(* IEC 61131-3 sources: std_i2980_v2.06_cp053/Source/IMM/ieccontrol/GlobalBaseArchives (part 4) *)

(* ---- FBGetRequiredPumps.pu ---- *)
(*
@h    ! WARNING !
@h    The Kemro K2 system (including software) only meets category B according to EN 954-1,
@h    thus it is not intended for usage in safety-relevant control applications in the field
@h    of personal safety (e.g. emergency stop).
@h    To implement potentially necessary safety-relevant control tasks, always use additional
@h    external safety devices that are intended for the particular purpose, and meet the necessary
@h    functional safety.
@h    For further information see EN 954-1 (EN ISO 13849-1) and/or the K2-x00 user manual, chapter
@h    "CE conformity, directives and standards".

get reference to the systemvariable with information about reuqired pumps for a defined movement
If the movement is not found, the reference pPumps is EMPTY.
*)

IMPORT_OVER_LISTFILE
 tsDeviceId
, tMoveIdent
, tsRequiredPumps
, tDeviceMovementList

END_IMPORT

FUNCTION_BLOCK FBGetRequiredPumps #DUMMY_EDIT_BLOCK

VAR_INPUT
 DeviceId : tsDeviceId;
 MoveDir : tMoveIdent;
 MoveId : tMoveIdent;
END_VAR

VAR_OUTPUT
 pPumps : REFTO tsRequiredPumps;
END_VAR

SYSTEM_VAR
 sv_DeviceMovements : tDeviceMovementList;
END_VAR

VAR_TEMP
 i : DINT;
 k : DINT;
END_VAR
#BEGIN_EDIT_BLOCK
(**************************************** WARNING ********************************************
 *** The KEBA Kemro K2 System including software is not intended for safety control tasks! ***
 ***                       For further information see Comment tab!                        ***
 *********************************************************************************************)

pPumps := EMPTY;

FOR i := 1 TO cMaxMoveDevicesRegistered DO
   IF (sv_DeviceMovements[i].DeviceId = DeviceId) THEN
      FOR k := 1 TO sv_DeviceMovements[i].iNumberOfMovements DO
         IF (sv_DeviceMovements[i].Movements[k]^.MoveDir = MoveDir) AND (sv_DeviceMovements[i].Movements[k]^.MoveId = MoveId) THEN
            pPumps := sv_DeviceMovements[i].Movements[k]^.AnaOutData.pRequiredPumps;
            EXIT;
         END_IF;
      END_FOR;
      EXIT;
   END_IF;
END_FOR;

;#END_EDIT_BLOCK END_FUNCTION_BLOCK

#END_OF_IEC_PART

@Puma @IecEditor 6 144 @Pou 25
@@@BEG_Comment@@@
@h    ! WARNING !
@h    The Kemro K2 system (including software) only meets category B according to EN 954-1,
@h    thus it is not intended for usage in safety-relevant control applications in the field
@h    of personal safety (e.g. emergency stop).
@h    To implement potentially necessary safety-relevant control tasks, always use additional
@h    external safety devices that are intended for the particular purpose, and meet the necessary
@h    functional safety.
@h    For further information see EN 954-1 (EN ISO 13849-1) and/or the K2-x00 user manual, chapter
@h    "CE conformity, directives and standards".

get reference to the systemvariable with information about reuqired pumps for a defined movement
If the movement is not found, the reference pPumps is EMPTY.
@@@END_Comment@@@

@BEG_Contents

@BEG_Func
@RT(17)FuncTreeContainer
0
@END_Func

@BEG_Const
@RT(18)ConstTreeContainer
0
@END_Const

@BEG_Export

@BEG_Kind
@FUNCTION_BLOCK @RT(18)FBGetRequiredPumps @STRUCTURED_TEXT
@RT(0) @RT(0) @RT(0)
@END_Kind

@BEG_Dcl
@RT(16)DclTreeContainer
7
@Var @RT(8)DeviceId @RT(0) @T @T @DERIVED 0 @T @T @DT @RT(10)tsDeviceId @RT(0) @T @T @UNKNOWN 0 @F
@F @F
@T
@BEG_Attrib
3 @RT(0) @RT(0) @RT(0)
@END_Attrib
1 1 @F @F @F @F

@Var @RT(7)MoveDir @RT(0) @T @T @DERIVED 0 @T @T @DT @RT(10)tMoveIdent @RT(0) @T @T @UNKNOWN 0 @F
@F @F
@T
@BEG_Attrib
3 @RT(0) @RT(0) @RT(0)
@END_Attrib
1 1 @F @F @F @F

@Var @RT(6)MoveId @RT(0) @T @T @DERIVED 0 @T @T @DT @RT(10)tMoveIdent @RT(0) @T @T @UNKNOWN 0 @F
@F @F
@T
@BEG_Attrib
3 @RT(0) @RT(0) @RT(0)
@END_Attrib
1 1 @F @F @F @F

@Var @RT(6)pPumps @RT(0) @T @T @REFTO 0 @F @DERIVED 0 @T @T @DT @RT(15)tsRequiredPumps @RT(0) @T @T @UNKNOWN 0 @F
@F @F
@T
@BEG_Attrib
3 @RT(0) @RT(0) @RT(0)
@END_Attrib
1 3 @F @F @F @F

@Var @RT(18)sv_DeviceMovements @RT(0) @T @T @DERIVED 0 @T @T @DT @RT(19)tDeviceMovementList @RT(0) @T @T @UNKNOWN 0 @F
@F @F
@T
@BEG_Attrib
3 @RT(0) @RT(0) @RT(0)
@END_Attrib
1 8 @F @F @F @F

@Var @RT(1)i @RT(0) @T @F @DT @RT(4)DINT @RT(0) @T @T @BASIC 0 @F
@F @F
@T
@BEG_Attrib
3 @RT(0) @RT(0) @RT(0)
@END_Attrib
1 4 @F @F @F @F

@Var @RT(1)k @RT(0) @T @F @DT @RT(4)DINT @RT(0) @T @T @BASIC 0 @F
@F @F
@T
@BEG_Attrib
3 @RT(0) @RT(0) @RT(0)
@END_Attrib
1 4 @F @F @F @F

@END_Dcl

@END_Export

@BEG_Body
@TL(20)
(**************************************** WARNING ********************************************
 *** The KEBA Kemro K2 System including software is not intended for safety control tasks! ***
 ***                       For further information see Comment tab!                        ***
 *********************************************************************************************)

pPumps := EMPTY;

FOR i := 1 TO cMaxMoveDevicesRegistered DO
   IF (sv_DeviceMovements[i].DeviceId = DeviceId) THEN
      FOR k := 1 TO sv_DeviceMovements[i].iNumberOfMovements DO
         IF (sv_DeviceMovements[i].Movements[k]^.MoveDir = MoveDir) AND (sv_DeviceMovements[i].Movements[k]^.MoveId = MoveId) THEN
            pPumps := sv_DeviceMovements[i].Movements[k]^.AnaOutData.pRequiredPumps;
            EXIT;
         END_IF;
      END_FOR;
      EXIT;
   END_IF;
END_FOR;

@END_Body

@END_Contents

(* ---- FBInitServoValveControlData.pu ---- *)
IMPORT_OVER_LISTFILE
 KAPPL_ServoValveControlData
, tsCylinderData
, KAPPL_ServoValveControllerMode
, tsVelPre
, tsControlParameters

END_IMPORT

FUNCTION_BLOCK FBInitServoValveControlData #DUMMY_EDIT_BLOCK

VAR_IN_OUT
 sServoValveControlData : KAPPL_ServoValveControlData;
END_VAR

VAR_INPUT
 pCylinderData : REFTO tsCylinderData;
 pCylinderStroke : REFTO REAL;
 pActPressureA : REFTO REAL;
 pSetPressureA : REFTO REAL;
 pSysPressure : REFTO REAL;
 pActPosition : REFTO REAL;
 pActVelocity : REFTO REAL;
 pSetVelocity : REFTO REAL;
 pControllerMode : REFTO KAPPL_ServoValveControllerMode;
 pTransducerError : REFTO BOOL;
 pConstSetupFwd : REFTO tsVelPre;
 pConstSetupBwd : REFTO tsVelPre;
 pDeviceReady : REFTO BOOL;
 pScrewDiameter : REFTO REAL;
 pMaxSpeedFwdMachLimit : REFTO REAL;
 pSetValueLimitActive : REFTO BOOL;
 pPressureControlParams : REFTO tsControlParameters;
 pBackPressureControlParams : REFTO tsControlParameters;
 pbMoveToServoCalibStartPos : REFTO BOOL;
END_VAR
#BEGIN_EDIT_BLOCK
sServoValveControlData.pCylinderData := pCylinderData;
sServoValveControlData.pCylinderStroke := pCylinderStroke;
sServoValveControlData.pActPressureA := pActPressureA;
sServoValveControlData.pSysPressure := pSysPressure;
sServoValveControlData.pActPosition := pActPosition;
sServoValveControlData.pActVelocity := pActVelocity;
sServoValveControlData.pControllerMode := pControllerMode;
sServoValveControlData.pTransducerError := pTransducerError;
sServoValveControlData.pConstSetupFwd := pConstSetupFwd;
sServoValveControlData.pConstSetupBwd := pConstSetupBwd;
sServoValveControlData.pSetPressureA := pSetPressureA;
sServoValveControlData.pSetVelocity := pSetVelocity;
sServoValveControlData.pDeviceReady := pDeviceReady;
sServoValveControlData.pScrewDiameter := pScrewDiameter;
sServoValveControlData.prMaxSpeedFwdMachLimit := pMaxSpeedFwdMachLimit;
sServoValveControlData.pSetValueLimitActive := pSetValueLimitActive;
sServoValveControlData.pPressureControlParams := pPressureControlParams;
sServoValveControlData.pBackPressureControlParams := pBackPressureControlParams;
sServoValveControlData.pbMoveToServoCalibStartPos := pbMoveToServoCalibStartPos;

;#END_EDIT_BLOCK END_FUNCTION_BLOCK

#END_OF_IEC_PART

@Puma @IecEditor 6 103 @Pou 25
@@@BEG_Comment@@@

@@@END_Comment@@@

@BEG_Contents

@BEG_Func
@RT(17)FuncTreeContainer
0
@END_Func

@BEG_Const
@RT(18)ConstTreeContainer
0
@END_Const

@BEG_Export

@BEG_Kind
@FUNCTION_BLOCK @RT(27)FBInitServoValveControlData @STRUCTURED_TEXT
@RT(0) @RT(0) @RT(0)
@END_Kind

@BEG_Dcl
@RT(16)DclTreeContainer
20
@Var @RT(22)sServoValveControlData @RT(0) @T @T @DERIVED 0 @T @T @DT @RT(27)KAPPL_ServoValveControlData @RT(0) @T @T @UNKNOWN 0 @F
@F @F
@T
@BEG_Attrib
3 @RT(0) @RT(0) @RT(0)
@END_Attrib
1 2 @F @F @F @F

@Var @RT(13)pCylinderData @RT(0) @T @T @REFTO 0 @F @DERIVED 0 @T @T @DT @RT(14)tsCylinderData @RT(0) @T @T @UNKNOWN 0 @F
@F @F
@T
@BEG_Attrib
3 @RT(0) @RT(0) @RT(0)
@END_Attrib
1 1 @F @F @F @F

@Var @RT(15)pCylinderStroke @RT(0) @T @T @REFTO 0 @T @DT @RT(4)REAL @RT(0) @T @T @BASIC 0 @F
@F @F
@T
@BEG_Attrib
3 @RT(0) @RT(0) @RT(0)
@END_Attrib
1 1 @F @F @F @F

@Var @RT(13)pActPressureA @RT(0) @T @T @REFTO 0 @T @DT @RT(4)REAL @RT(0) @T @T @BASIC 0 @F
@F @F
@T
@BEG_Attrib
3 @RT(0) @RT(0) @RT(0)
@END_Attrib
1 1 @F @F @F @F

@Var @RT(13)pSetPressureA @RT(0) @T @T @REFTO 0 @T @DT @RT(4)REAL @RT(0) @T @T @BASIC 0 @F
@F @F
@T
@BEG_Attrib
3 @RT(0) @RT(0) @RT(0)
@END_Attrib
1 1 @F @F @F @F

@Var @RT(12)pSysPressure @RT(0) @T @T @REFTO 0 @T @DT @RT(4)REAL @RT(0) @T @T @BASIC 0 @F
@F @F
@T
@BEG_Attrib
3 @RT(0) @RT(0) @RT(0)
@END_Attrib
1 1 @F @F @F @F

@Var @RT(12)pActPosition @RT(0) @T @T @REFTO 0 @T @DT @RT(4)REAL @RT(0) @T @T @BASIC 0 @F
@F @F
@T
@BEG_Attrib
3 @RT(0) @RT(0) @RT(0)
@END_Attrib
1 1 @F @F @F @F

@Var @RT(12)pActVelocity @RT(0) @T @T @REFTO 0 @T @DT @RT(4)REAL @RT(0) @T @T @BASIC 0 @F
@F @F
@T
@BEG_Attrib
3 @RT(0) @RT(0) @RT(0)
@END_Attrib
1 1 @F @F @F @F

@Var @RT(12)pSetVelocity @RT(0) @T @T @REFTO 0 @T @DT @RT(4)REAL @RT(0) @T @T @BASIC 0 @F
@F @F
@T
@BEG_Attrib
3 @RT(0) @RT(0) @RT(0)
@END_Attrib
1 1 @F @F @F @F

@Var @RT(15)pControllerMode @RT(0) @T @T @REFTO 0 @F @DERIVED 0 @T @T @DT @RT(30)KAPPL_ServoValveControllerMode @RT(0) @T @T @UNKNOWN 0 @F
@F @F
@T
@BEG_Attrib
3 @RT(0) @RT(0) @RT(0)
@END_Attrib
1 1 @F @F @F @F

@Var @RT(16)pTransducerError @RT(0) @T @T @REFTO 0 @T @DT @RT(4)BOOL @RT(0) @T @T @BASIC 0 @F
@F @F
@T
@BEG_Attrib
3 @RT(0) @RT(0) @RT(0)
@END_Attrib
1 1 @F @F @F @F

@Var @RT(14)pConstSetupFwd @RT(0) @T @T @REFTO 0 @F @DERIVED 0 @T @T @DT @RT(8)tsVelPre @RT(0) @T @T @UNKNOWN 0 @F
@F @F
@T
@BEG_Attrib
3 @RT(0) @RT(0) @RT(0)
@END_Attrib
1 1 @F @F @F @F

@Var @RT(14)pConstSetupBwd @RT(0) @T @T @REFTO 0 @F @DERIVED 0 @T @T @DT @RT(8)tsVelPre @RT(0) @T @T @UNKNOWN 0 @F
@F @F
@T
@BEG_Attrib
3 @RT(0) @RT(0) @RT(0)
@END_Attrib
1 1 @F @F @F @F

@Var @RT(12)pDeviceReady @RT(0) @T @T @REFTO 0 @T @DT @RT(4)BOOL @RT(0) @T @T @BASIC 0 @F
@F @F
@T
@BEG_Attrib
3 @RT(0) @RT(0) @RT(0)
@END_Attrib
1 1 @F @F @F @F

@Var @RT(14)pScrewDiameter @RT(0) @T @T @REFTO 0 @T @DT @RT(4)REAL @RT(0) @T @T @BASIC 0 @F
@F @F
@T
@BEG_Attrib
3 @RT(0) @RT(0) @RT(0)
@END_Attrib
1 1 @F @F @F @F

@Var @RT(21)pMaxSpeedFwdMachLimit @RT(0) @T @T @REFTO 0 @T @DT @RT(4)REAL @RT(0) @T @T @BASIC 0 @F
@F @F
@T
@BEG_Attrib
3 @RT(0) @RT(0) @RT(0)
@END_Attrib
1 1 @F @F @F @F

@Var @RT(20)pSetValueLimitActive @RT(0) @T @T @REFTO 0 @T @DT @RT(4)BOOL @RT(0) @T @T @BASIC 0 @F
@F @F
@T
@BEG_Attrib
3 @RT(0) @RT(0) @RT(0)
@END_Attrib
1 1 @F @F @F @F

@Var @RT(22)pPressureControlParams @RT(0) @T @T @REFTO 0 @F @DERIVED 0 @T @T @DT @RT(19)tsControlParameters @RT(0) @T @T @UNKNOWN 0 @F
@F @F
@T
@BEG_Attrib
3 @RT(0) @RT(0) @RT(0)
@END_Attrib
1 1 @F @F @F @F

@Var @RT(26)pBackPressureControlParams @RT(0) @T @T @REFTO 0 @F @DERIVED 0 @T @T @DT @RT(19)tsControlParameters @RT(0) @T @T @UNKNOWN 0 @F
@F @F
@T
@BEG_Attrib
3 @RT(0) @RT(0) @RT(0)
@END_Attrib
1 1 @F @F @F @F

@Var @RT(26)pbMoveToServoCalibStartPos @RT(0) @T @T @REFTO 0 @T @DT @RT(4)BOOL @RT(0) @T @T @BASIC 0 @F
@F @F
@T
@BEG_Attrib
3 @RT(0) @RT(0) @RT(0)
@END_Attrib
1 1 @F @F @F @F

@END_Dcl

@END_Export

@BEG_Body
@TL(21)
sServoValveControlData.pCylinderData := pCylinderData;
sServoValveControlData.pCylinderStroke := pCylinderStroke;
sServoValveControlData.pActPressureA := pActPressureA;
sServoValveControlData.pSysPressure := pSysPressure;
sServoValveControlData.pActPosition := pActPosition;
sServoValveControlData.pActVelocity := pActVelocity;
sServoValveControlData.pControllerMode := pControllerMode;
sServoValveControlData.pTransducerError := pTransducerError;
sServoValveControlData.pConstSetupFwd := pConstSetupFwd;
sServoValveControlData.pConstSetupBwd := pConstSetupBwd;
sServoValveControlData.pSetPressureA := pSetPressureA;
sServoValveControlData.pSetVelocity := pSetVelocity;
sServoValveControlData.pDeviceReady := pDeviceReady;
sServoValveControlData.pScrewDiameter := pScrewDiameter;
sServoValveControlData.prMaxSpeedFwdMachLimit := pMaxSpeedFwdMachLimit;
sServoValveControlData.pSetValueLimitActive := pSetValueLimitActive;
sServoValveControlData.pPressureControlParams := pPressureControlParams;
sServoValveControlData.pBackPressureControlParams := pBackPressureControlParams;
sServoValveControlData.pbMoveToServoCalibStartPos := pbMoveToServoCalibStartPos;

@END_Body

@END_Contents

(* ---- FBLintabCopy.pu ---- *)
(*
 /*-------------------------------------------------------------------------
 *                   (c) 2002 by KEBA Ges.m.b.H & Co
 *                            Linz/AUSTRIA
 *                         All rights reserved
 *--------------------------------------------------------------------------
 *    Projekt   : KEMRO.appl.2.plastics
 *    Erstautor : prg
 *    Datum     : 20.02.2003
 *    $Author: Admin $
 *    $Revision: 8 $
 *    $Modtime: 4.07.07 11:02 $
 *    $Archive: /ApplicationFrames/KePlast/APPL/ApplMoldMachineIECLib_Servo/FBPreCutOff.pu $
 *--------------------------------------------------------------------------*/
*)

IMPORT_OVER_LISTFILE
 cApplPlasticsWrongPIDParams
, cApplPlasticsPIDCalcFailed
, cApplPlasticsNoError
, KAPPL_LintabData
, tLintabPoints
//  KCTRL_LintabPoints

END_IMPORT

FUNCTION_BLOCK FBLintabCopy #DUMMY_EDIT_BLOCK

VAR_INPUT
 LintabLight : REFTO KAPPL_LintabData (* Start pre injection movement *);
 LintabRef : REFTO tLintabPoints;
END_VAR

// VAR_OUTPUT
 // Lintab : KCTRL_LintabPoints (* Cycletime of calling task *);
// END_VAR

VAR
 LintabHelp : REFTO tLintabPoints;
 uCount : UDINT;
 float : REAL;
END_VAR
#BEGIN_EDIT_BLOCK
//Lintab.uNoOfPoints := LintabLight^ .LintabPoints.uNoOfPoints;
LintabHelp := LintabRef;
FOR uCount :=1 TO LintabLight^ .LintabPoints.uNoOfPoints DO
   LintabHelp^[uCount].rX := LintabLight^.LintabPoints.Point[uCount].rX;
   LintabHelp^[uCount].rY := LintabLight^.LintabPoints.Point[uCount].rY;
END_FOR;

;#END_EDIT_BLOCK END_FUNCTION_BLOCK

#END_OF_IEC_PART

@Puma @IecEditor 6 68 @Pou 25
@@@BEG_Comment@@@
 /*-------------------------------------------------------------------------
 *                   (c) 2002 by KEBA Ges.m.b.H & Co
 *                            Linz/AUSTRIA
 *                         All rights reserved
 *--------------------------------------------------------------------------
 *    Projekt   : KEMRO.appl.2.plastics
 *    Erstautor : prg
 *    Datum     : 20.02.2003
 *    $Author: Admin $
 *    $Revision: 8 $
 *    $Modtime: 4.07.07 11:02 $
 *    $Archive: /ApplicationFrames/KePlast/APPL/ApplMoldMachineIECLib_Servo/FBPreCutOff.pu $
 *--------------------------------------------------------------------------*/
@@@END_Comment@@@

@BEG_Contents

@BEG_Func
@RT(17)FuncTreeContainer
0
@END_Func

@BEG_Const
@RT(18)ConstTreeContainer
3
@Var @RT(27)cApplPlasticsWrongPIDParams @RT(0) @T @F @DT @RT(4)DINT @RT(0) @T @T @BASIC 0 @F
@F @F
@T
@BEG_Attrib
0 @RT(4)-151 @RT(51)PID - regulator params are wrong or not initialized
@END_Attrib
1 1 @F @F @F @F

@Var @RT(26)cApplPlasticsPIDCalcFailed @RT(0) @T @F @DT @RT(4)DINT @RT(0) @T @T @BASIC 0 @F
@F @F
@T
@BEG_Attrib
0 @RT(4)-152 @RT(29)cyclic PID calculation failed
@END_Attrib
1 1 @F @F @F @F

@Var @RT(20)cApplPlasticsNoError @RT(0) @T @F @DT @RT(4)DINT @RT(0) @T @T @BASIC 0 @F
@F @F
@T
@BEG_Attrib
0 @RT(1)0 @RT(8)No Error
@END_Attrib
1 1 @F @F @F @F

@END_Const

@BEG_Export

@BEG_Kind
@FUNCTION_BLOCK @RT(12)FBLintabCopy @STRUCTURED_TEXT
@RT(0) @RT(0) @RT(0)
@END_Kind

@BEG_Dcl
@RT(16)DclTreeContainer
6
@Var @RT(11)LintabLight @RT(0) @T @T @REFTO 0 @F @DERIVED 0 @T @T @DT @RT(16)KAPPL_LintabData @RT(0) @T @T @UNKNOWN 0 @F
@F @F
@T
@BEG_Attrib
3 @RT(0) @RT(28)Start pre injection movement @RT(0)
@END_Attrib
1 1 @F @F @F @F

@Var @RT(9)LintabRef @RT(0) @T @T @REFTO 0 @F @DERIVED 0 @T @T @DT @RT(13)tLintabPoints @RT(0) @T @T @UNKNOWN 0 @F
@F @F
@T
@BEG_Attrib
3 @RT(0) @RT(0) @RT(0)
@END_Attrib
1 1 @F @F @F @F

@Var @RT(10)LintabHelp @RT(0) @T @T @REFTO 0 @F @DERIVED 0 @T @T @DT @RT(13)tLintabPoints @RT(0) @T @T @UNKNOWN 0 @F
@F @F
@T
@BEG_Attrib
3 @RT(0) @RT(0) @RT(0)
@END_Attrib
1 0 @F @F @F @F

@Var @RT(6)Lintab @RT(0) @T @T @DERIVED 0 @T @T @DT @RT(18)KCTRL_LintabPoints @RT(0) @T @T @UNKNOWN 0 @F
@F @T
@T
@BEG_Attrib
3 @RT(0) @RT(25)Cycletime of calling task @RT(0)
@END_Attrib
1 3 @F @F @F @F

@Var @RT(6)uCount @RT(0) @T @F @DT @RT(5)UDINT @RT(0) @T @T @BASIC 0 @F
@F @F
@T
@BEG_Attrib
3 @RT(0) @RT(0) @RT(0)
@END_Attrib
1 0 @F @F @F @F

@Var @RT(5)float @RT(0) @T @F @DT @RT(4)REAL @RT(0) @T @T @BASIC 0 @F
@F @F
@T
@BEG_Attrib
3 @RT(0) @RT(0) @RT(0)
@END_Attrib
1 0 @F @F @F @F

@END_Dcl

@END_Export

@BEG_Body
@TL(7)
//Lintab.uNoOfPoints := LintabLight^ .LintabPoints.uNoOfPoints;
LintabHelp := LintabRef;
FOR uCount :=1 TO LintabLight^ .LintabPoints.uNoOfPoints DO
   LintabHelp^[uCount].rX := LintabLight^.LintabPoints.Point[uCount].rX;
   LintabHelp^[uCount].rY := LintabLight^.LintabPoints.Point[uCount].rY;
END_FOR;

@END_Body

@END_Contents

(* ---- FBLockUnlock.pu ---- *)
(*
This FunktionBlock locks a specified Movement.
Movements can be locked or unlocked every time, no matter if the movement is active or inactive.
With the parameter "Mode" 2 different Lock-Modes and the Unlock-Mode can be chosen.

Mode = enLockResume
  -if an inactive movement is locked and started afterwards it will stand still until it is being unlocked.
  -if an active movement is being locked it stopps its motion until it is being unlocked.
  In both cases the movement resumes its motion automatically after unlocking.

Mode = enLockAbort
  -if an inactively locked movement is tried to be started it will inactively remain until it is being unlocked and started again.
  -if an active movement is being locked it will stop its motion. To restart the movement it has to be unlocked first
   and started again.

Mode = Unlock
   Unlock Movement

All Components of the system can be locked by DeviceId.CompId := cCompAll
All Devices of a component can be locked by DeviceId.IndexId := cAllDevIndex
*)

IMPORT_OVER_LISTFILE
 ASSERT
, tsDeviceId
, tMoveIdent
, tsAlarm
, tnLockUnlock
, tevLockUnlockData
, tevLockUnlock

END_IMPORT

FUNCTION_BLOCK FBLockUnlock #DUMMY_EDIT_BLOCK

VAR_INPUT
 DeviceId : tsDeviceId (* Device which should be locked *);
 MoveDir : tMoveIdent (* Movement direction to lock *);
 MoveId : tMoveIdent (* Movement ID to lock *);
 Alarm : tsAlarm (* Alarm that is set if the locked movement is tried to be started *);
 Mode : tnLockUnlock (* Modes: enLockResume, enLockAbort, enUnlock *);
 bSetAlarmImmediately : BOOL (* FALSE: alarm is set if locked movement should be started; TRUE: alarm is set immediately *);
END_VAR

SYSTEM_VAR
 sv_DeviceId : tsDeviceId;
 sv_bInitDone : BOOL;
END_VAR

SYSTEM_OBJECT
 evLockUnlock : tevLockUnlock;
 erAssert : ALARM;
END_OBJECT

VAR
 evLockUnlockData : tevLockUnlockData;
 dummy : BOOL;
END_VAR
#BEGIN_EDIT_BLOCK
(**************************************** WARNING ********************************************
 *** The KEBA Kemro K2 System including software is not intended for safety control tasks! ***
 ***                       For further information see Comment tab!                        ***
 *********************************************************************************************)

//if the movements are still not registered, gives application programmer code offset and frame offset
dummy := ASSERT(sv_bInitDone, erAssert);

evLockUnlockData.DeviceId       := DeviceId;
evLockUnlockData.DeviceIdSender := sv_DeviceId;
evLockUnlockData.MoveDir        := MoveDir;
evLockUnlockData.MoveId         := MoveId;
evLockUnlockData.Alarm          := Alarm;
evLockUnlockData.Mode           := Mode;
evLockUnlockData.bSetAlarmImmediately := bSetAlarmImmediately;
SET_EVENT(evLockUnlock, evLockUnlockData);

;#END_EDIT_BLOCK END_FUNCTION_BLOCK

#END_OF_IEC_PART

@Puma @IecEditor 6 10 @Pou 25
@@@BEG_Comment@@@
This FunktionBlock locks a specified Movement.
Movements can be locked or unlocked every time, no matter if the movement is active or inactive.
With the parameter "Mode" 2 different Lock-Modes and the Unlock-Mode can be chosen.

Mode = enLockResume
  -if an inactive movement is locked and started afterwards it will stand still until it is being unlocked.
  -if an active movement is being locked it stopps its motion until it is being unlocked.
  In both cases the movement resumes its motion automatically after unlocking.

Mode = enLockAbort
  -if an inactively locked movement is tried to be started it will inactively remain until it is being unlocked and started again.
  -if an active movement is being locked it will stop its motion. To restart the movement it has to be unlocked first
   and started again.

Mode = Unlock
   Unlock Movement

All Components of the system can be locked by DeviceId.CompId := cCompAll
All Devices of a component can be locked by DeviceId.IndexId := cAllDevIndex
@@@END_Comment@@@

@BEG_Contents

@BEG_Func
@RT(17)FuncTreeContainer
1
@Var @RT(6)ASSERT @RT(0) @T @T @DERIVED 0 @F @RT(8)FUNCTION @F
@T
@BEG_Attrib
0 @RT(0) @RT(0)
@END_Attrib
1 1 @F @F @F @F

@END_Func

@BEG_Const
@RT(18)ConstTreeContainer
0
@END_Const

@BEG_Export

@BEG_Kind
@FUNCTION_BLOCK @RT(12)FBLockUnlock @STRUCTURED_TEXT
@RT(0) @RT(0) @RT(0)
@END_Kind

@BEG_Dcl
@RT(16)DclTreeContainer
12
@Var @RT(8)DeviceId @RT(0) @T @T @DERIVED 0 @T @T @DT @RT(10)tsDeviceId @RT(0) @T @T @UNKNOWN 0 @F
@F @F
@T
@BEG_Attrib
3 @RT(0) @RT(29)Device which should be locked @RT(0)
@END_Attrib
1 1 @F @F @F @F

@Var @RT(7)MoveDir @RT(0) @T @T @DERIVED 0 @T @T @DT @RT(10)tMoveIdent @RT(0) @T @T @UNKNOWN 0 @F
@F @F
@T
@BEG_Attrib
3 @RT(0) @RT(26)Movement direction to lock @RT(0)
@END_Attrib
1 1 @F @F @F @F

@Var @RT(6)MoveId @RT(0) @T @T @DERIVED 0 @T @T @DT @RT(10)tMoveIdent @RT(0) @T @T @UNKNOWN 0 @F
@F @F
@T
@BEG_Attrib
3 @RT(0) @RT(19)Movement ID to lock @RT(0)
@END_Attrib
1 1 @F @F @F @F

@Var @RT(5)Alarm @RT(0) @T @T @DERIVED 0 @T @T @DT @RT(7)tsAlarm @RT(0) @T @T @UNKNOWN 0 @F
@F @F
@T
@BEG_Attrib
3 @RT(0) @RT(63)Alarm that is set if the locked movement is tried to be started @RT(0)
@END_Attrib
1 1 @F @F @F @F

@Var @RT(4)Mode @RT(0) @T @T @DERIVED 0 @T @T @DT @RT(12)tnLockUnlock @RT(0) @T @T @UNKNOWN 0 @F
@F @F
@T
@BEG_Attrib
3 @RT(0) @RT(42)Modes: enLockResume, enLockAbort, enUnlock @RT(0)
@END_Attrib
1 1 @F @F @F @F

@Var @RT(16)evLockUnlockData @RT(0) @T @T @DERIVED 0 @T @T @DT @RT(17)tevLockUnlockData @RT(0) @T @T @UNKNOWN 0 @F
@F @F
@T
@BEG_Attrib
3 @RT(0) @RT(0) @RT(0)
@END_Attrib
1 0 @F @F @F @F

@Var @RT(12)evLockUnlock @RT(0) @T @T @DERIVED 0 @T @T @DT @RT(13)tevLockUnlock @RT(0) @T @T @UNKNOWN 0 @F
@F @F
@T
@BEG_Attrib
3 @RT(0) @RT(0) @RT(0)
@END_Attrib
1 7 @F @F @F @F

@Var @RT(11)sv_DeviceId @RT(0) @T @T @DERIVED 0 @T @T @DT @RT(10)tsDeviceId @RT(0) @T @T @UNKNOWN 0 @F
@F @F
@T
@BEG_Attrib
3 @RT(0) @RT(0) @RT(0)
@END_Attrib
1 8 @F @F @F @F

@Var @RT(8)erAssert @RT(0) @T @F @DT @RT(5)ALARM @RT(0) @T @T @BASIC 0 @F
@F @F
@T
@BEG_Attrib
3 @RT(0) @RT(0) @RT(0)
@END_Attrib
1 7 @F @F @F @F

@Var @RT(5)dummy @RT(0) @T @F @DT @RT(4)BOOL @RT(0) @T @T @BASIC 0 @F
@F @F
@T
@BEG_Attrib
3 @RT(0) @RT(0) @RT(0)
@END_Attrib
1 0 @F @F @F @F

@Var @RT(12)sv_bInitDone @RT(0) @T @F @DT @RT(4)BOOL @RT(0) @T @T @BASIC 0 @F
@F @F
@T
@BEG_Attrib
3 @RT(0) @RT(0) @RT(0)
@END_Attrib
1 8 @F @F @F @F

@Var @RT(20)bSetAlarmImmediately @RT(0) @T @F @DT @RT(4)BOOL @RT(0) @T @T @BASIC 0 @F
@F @F
@T
@BEG_Attrib
3 @RT(0) @RT(88)FALSE: alarm is set if locked movement should be started; TRUE: alarm is set immediately @RT(0)
@END_Attrib
1 1 @F @F @F @F

@END_Dcl

@END_Export

@BEG_Body
@TL(17)
(**************************************** WARNING ********************************************
 *** The KEBA Kemro K2 System including software is not intended for safety control tasks! ***
 ***                       For further information see Comment tab!                        ***
 *********************************************************************************************)

//if the movements are still not registered, gives application programmer code offset and frame offset
dummy := ASSERT(sv_bInitDone, erAssert);

evLockUnlockData.DeviceId       := DeviceId;
evLockUnlockData.DeviceIdSender := sv_DeviceId;
evLockUnlockData.MoveDir        := MoveDir;
evLockUnlockData.MoveId         := MoveId;
evLockUnlockData.Alarm          := Alarm;
evLockUnlockData.Mode           := Mode;
evLockUnlockData.bSetAlarmImmediately := bSetAlarmImmediately;
SET_EVENT(evLockUnlock, evLockUnlockData);

@END_Body

@END_Contents

(* ---- FBLockUnlockGroup.pu ---- *)
(*
With this FunctionBlock a group of movements can be locked.
Groups can be locked or unlocked every time, no matter if a member of the group is active or inactive.
With the parameter "Mode" 2 different Lock-Modes and the Unlock-Mode can be chosen.

Mode = enLockResume
  -if an inactive movement is locked and started afterwards it will stand still until it is being unlocked.
  -if an active movement is being locked it stopps its motion until it is being unlocked.
  In both cases the movement resumes its motion automatically after unlocking.

Mode = enLockAbort
  -if an inactively locked movement is tried to be started it will inactively remain until it is being unlocked and started again.
  -if an active movement is being locked it will stop its motion. To restart the movement it has to be unlocked first
   and started again.

Mode = Unlock
   Unlock Movement

The group-membership of each movement has to be defined in systemVariable sv_MoveXxx.LockGroups[].
Every movement can be member of multible lockgroups.
The lockgroups itself are defined by constants in the LockGroups.tu file
*)

IMPORT_OVER_LISTFILE
 ASSERT
, tLockGroup
, tsAlarm
, tnLockUnlock
, tevLockUnlockGroup
, tevLockUnlockGroupData
, tsDeviceId

END_IMPORT

FUNCTION_BLOCK FBLockUnlockGroup #DUMMY_EDIT_BLOCK

VAR_INPUT
 Group : tLockGroup (* Group to lock *);
 Alarm : tsAlarm (* this alarm is set if the locked movement is tried to be started *);
 Mode : tnLockUnlock (* Modes: enLockResume, enLockAbort, enUnlock *);
 bSetAlarmImmediately : BOOL (* FALSE: alarm is set if locked movement should be started; TRUE: alarm is set immediately *);
END_VAR

SYSTEM_VAR
 sv_DeviceId : tsDeviceId;
 sv_bInitDone : BOOL;
END_VAR

SYSTEM_OBJECT
 evLockUnlockGroup : tevLockUnlockGroup;
 erAssert : ALARM;
END_OBJECT

VAR
 evLockUnlockGroupData : tevLockUnlockGroupData;
 dummy : BOOL;
END_VAR
#BEGIN_EDIT_BLOCK
(**************************************** WARNING ********************************************
 *** The KEBA Kemro K2 System including software is not intended for safety control tasks! ***
 ***                       For further information see Comment tab!                        ***
 *********************************************************************************************)

//if the movements are still not registered, gives application programmer code offset and frame offset
dummy := ASSERT(sv_bInitDone, erAssert);

evLockUnlockGroupData.DeviceIdSender := sv_DeviceId;
evLockUnlockGroupData.Group          := Group;
evLockUnlockGroupData.Alarm          := Alarm;
evLockUnlockGroupData.Mode           := Mode;
evLockUnlockGroupData.bSetAlarmImmediately := bSetAlarmImmediately;
SET_EVENT(evLockUnlockGroup, evLockUnlockGroupData);

;#END_EDIT_BLOCK END_FUNCTION_BLOCK

#END_OF_IEC_PART

@Puma @IecEditor 6 10 @Pou 25
@@@BEG_Comment@@@
With this FunctionBlock a group of movements can be locked.
Groups can be locked or unlocked every time, no matter if a member of the group is active or inactive.
With the parameter "Mode" 2 different Lock-Modes and the Unlock-Mode can be chosen.

Mode = enLockResume
  -if an inactive movement is locked and started afterwards it will stand still until it is being unlocked.
  -if an active movement is being locked it stopps its motion until it is being unlocked.
  In both cases the movement resumes its motion automatically after unlocking.

Mode = enLockAbort
  -if an inactively locked movement is tried to be started it will inactively remain until it is being unlocked and started again.
  -if an active movement is being locked it will stop its motion. To restart the movement it has to be unlocked first
   and started again.

Mode = Unlock
   Unlock Movement

The group-membership of each movement has to be defined in systemVariable sv_MoveXxx.LockGroups[].
Every movement can be member of multible lockgroups.
The lockgroups itself are defined by constants in the LockGroups.tu file
@@@END_Comment@@@

@BEG_Contents

@BEG_Func
@RT(17)FuncTreeContainer
1
@Var @RT(6)ASSERT @RT(0) @T @T @DERIVED 0 @F @RT(8)FUNCTION @F
@T
@BEG_Attrib
0 @RT(0) @RT(0)
@END_Attrib
1 1 @F @F @F @F

@END_Func

@BEG_Const
@RT(18)ConstTreeContainer
0
@END_Const

@BEG_Export

@BEG_Kind
@FUNCTION_BLOCK @RT(17)FBLockUnlockGroup @STRUCTURED_TEXT
@RT(0) @RT(0) @RT(0)
@END_Kind

@BEG_Dcl
@RT(16)DclTreeContainer
10
@Var @RT(5)Group @RT(0) @T @T @DERIVED 0 @T @T @DT @RT(10)tLockGroup @RT(0) @T @T @UNKNOWN 0 @F
@F @F
@T
@BEG_Attrib
3 @RT(0) @RT(13)Group to lock @RT(0)
@END_Attrib
1 1 @F @F @F @F

@Var @RT(5)Alarm @RT(0) @T @T @DERIVED 0 @T @T @DT @RT(7)tsAlarm @RT(0) @T @T @UNKNOWN 0 @F
@F @F
@T
@BEG_Attrib
3 @RT(0) @RT(63)this alarm is set if the locked movement is tried to be started @RT(0)
@END_Attrib
1 1 @F @F @F @F

@Var @RT(4)Mode @RT(0) @T @T @DERIVED 0 @T @T @DT @RT(12)tnLockUnlock @RT(0) @T @T @UNKNOWN 0 @F
@F @F
@T
@BEG_Attrib
3 @RT(0) @RT(42)Modes: enLockResume, enLockAbort, enUnlock @RT(0)
@END_Attrib
1 1 @F @F @F @F

@Var @RT(17)evLockUnlockGroup @RT(0) @T @T @DERIVED 0 @T @T @DT @RT(18)tevLockUnlockGroup @RT(0) @T @T @UNKNOWN 0 @F
@F @F
@T
@BEG_Attrib
3 @RT(0) @RT(0) @RT(0)
@END_Attrib
1 7 @F @F @F @F

@Var @RT(21)evLockUnlockGroupData @RT(0) @T @T @DERIVED 0 @T @T @DT @RT(22)tevLockUnlockGroupData @RT(0) @T @T @UNKNOWN 0 @F
@F @F
@T
@BEG_Attrib
3 @RT(0) @RT(0) @RT(0)
@END_Attrib
1 0 @F @F @F @F

@Var @RT(11)sv_DeviceId @RT(0) @T @T @DERIVED 0 @T @T @DT @RT(10)tsDeviceId @RT(0) @T @T @UNKNOWN 0 @F
@F @F
@T
@BEG_Attrib
3 @RT(0) @RT(0) @RT(0)
@END_Attrib
1 8 @F @F @F @F

@Var @RT(8)erAssert @RT(0) @T @F @DT @RT(5)ALARM @RT(0) @T @T @BASIC 0 @F
@F @F
@T
@BEG_Attrib
3 @RT(0) @RT(0) @RT(0)
@END_Attrib
1 7 @F @F @F @F

@Var @RT(5)dummy @RT(0) @T @F @DT @RT(4)BOOL @RT(0) @T @T @BASIC 0 @F
@F @F
@T
@BEG_Attrib
3 @RT(0) @RT(0) @RT(0)
@END_Attrib
1 0 @F @F @F @F

@Var @RT(12)sv_bInitDone @RT(0) @T @F @DT @RT(4)BOOL @RT(0) @T @T @BASIC 0 @F
@F @F
@T
@BEG_Attrib
3 @RT(0) @RT(0) @RT(0)
@END_Attrib
1 8 @F @F @F @F

@Var @RT(20)bSetAlarmImmediately @RT(0) @T @F @DT @RT(4)BOOL @RT(0) @T @T @BASIC 0 @F
@F @F
@T
@BEG_Attrib
3 @RT(0) @RT(88)FALSE: alarm is set if locked movement should be started; TRUE: alarm is set immediately @RT(0)
@END_Attrib
1 1 @F @F @F @F

@END_Dcl

@END_Export

@BEG_Body
@TL(15)
(**************************************** WARNING ********************************************
 *** The KEBA Kemro K2 System including software is not intended for safety control tasks! ***
 ***                       For further information see Comment tab!                        ***
 *********************************************************************************************)

//if the movements are still not registered, gives application programmer code offset and frame offset
dummy := ASSERT(sv_bInitDone, erAssert);

evLockUnlockGroupData.DeviceIdSender := sv_DeviceId;
evLockUnlockGroupData.Group          := Group;
evLockUnlockGroupData.Alarm          := Alarm;
evLockUnlockGroupData.Mode           := Mode;
evLockUnlockGroupData.bSetAlarmImmediately := bSetAlarmImmediately;
SET_EVENT(evLockUnlockGroup, evLockUnlockGroupData);

@END_Body

@END_Contents

(* ---- FBManualButton.pu ---- *)
(*
Send evStartRequest and evStopRequest events to start a manual movement with a button.

bButton should represent the actual state of the button
(pressed/released)

In half or full auto mode this block will not
react to button press/release
and thus will not send evStartRequest or evStopRequest events.

This FB has a non sticky behavior.
On button press start the movement.
On button release stop the movement.
*)

IMPORT_OVER_LISTFILE
 SET_EVENT
, nHalfAutomatic
, cMoveNone
, tMoveIdent
, tnOperationMode
, tsDeviceId
, tevStartRequest
, tevStopRequest
, tevStartRequestData
, tevStopRequestData

END_IMPORT

FUNCTION_BLOCK FBManualButton #DUMMY_EDIT_BLOCK

VAR_INPUT
 bButton : BOOL;
 MoveId : tMoveIdent;
 MoveDir : tMoveIdent;
 IntermediateCond : DINT;
END_VAR

SYSTEM_VAR
 sv_bDeviceReady : BOOL;
 sv_OperationMode : tnOperationMode;
 sv_DeviceId : tsDeviceId;
 sv_bAutoCalibRunning : BOOL;
 sv_bSequenceInterruption : BOOL (* TRUE: sequence is interrupted *);
END_VAR

SYSTEM_OBJECT
 evStartRequest : tevStartRequest;
 evStopRequest : tevStopRequest;
END_OBJECT

VAR
 ActiveMoveId : tMoveIdent;
 ActiveMoveDir : tMoveIdent;
 evStartRequestData : tevStartRequestData;
 evStopRequestData : tevStopRequestData;
END_VAR
#BEGIN_EDIT_BLOCK
(**************************************** WARNING ********************************************
 *** The KEBA Kemro K2 System including software is not intended for safety control tasks! ***
 ***                       For further information see Comment tab!                        ***
 *********************************************************************************************)

IF ((sv_OperationMode >= nHalfAutomatic) AND NOT sv_bSequenceInterruption) OR sv_bAutoCalibRunning THEN
   //do not react on manual buttons in half or fullauto mode or during active autocalibration
   //if sequence is interrupted, some movements are allowed
   RETURN;
END_IF;

IF MoveId > 0 AND
   MoveDir > 0 THEN

   // only start movement if butten is not currently running another movement
   IF bButton AND sv_bDeviceReady AND
      ActiveMoveDir = cMoveNone AND
      ActiveMoveId = cMoveNone THEN

      // remember active movement in case button is used for 2 different MoveID/MoveDir
      // so pressing the second button can not cause any problems
      ActiveMoveDir := MoveDir;
      ActiveMoveId := MoveId;

      // send start request
      evStartRequestData.DeviceId := sv_DeviceId;
      evStartRequestData.MoveDir := MoveDir;
      evStartRequestData.MoveId := MoveId;
      evStartRequestData.IntermediateCond := IntermediateCond;
      SET_EVENT(evStartRequest, evStartRequestData);

   END_IF;

   IF NOT bButton AND
      MoveDir = ActiveMoveDir AND
      MoveId  = ActiveMoveId THEN

      //stop Movement
      evStopRequestData.DeviceId := sv_DeviceId;
      evStopRequestData.MoveDir := ActiveMoveDir;
      evStopRequestData.MoveId := ActiveMoveId;
      SET_EVENT(evStopRequest, evStopRequestData);

      ActiveMoveDir := cMoveNone;
      ActiveMoveId := cMoveNone;
   END_IF;
END_IF;

;#END_EDIT_BLOCK END_FUNCTION_BLOCK

#END_OF_IEC_PART

@Puma @IecEditor 6 114 @Pou 25
@@@BEG_Comment@@@
Send evStartRequest and evStopRequest events to start a manual movement with a button.

bButton should represent the actual state of the button
(pressed/released)

In half or full auto mode this block will not
react to button press/release
and thus will not send evStartRequest or evStopRequest events.

This FB has a non sticky behavior.
On button press start the movement.
On button release stop the movement.
@@@END_Comment@@@

@BEG_Contents

@BEG_Func
@RT(17)FuncTreeContainer
1
@Var @RT(9)SET_EVENT @RT(0) @T @T @DERIVED 0 @F @RT(23)KEBA_STANDARD_PROCEDURE @F
@T
@BEG_Attrib
0 @RT(0) @RT(0)
@END_Attrib
1 1 @F @F @F @F

@END_Func

@BEG_Const
@RT(18)ConstTreeContainer
2
@Var @RT(14)nHalfAutomatic @RT(0) @T @T @DERIVED 0 @F @RT(15)tnOperationMode @F
@T
@BEG_Attrib
0 @RT(1)2 @RT(34)confirmation every cycle necessary
@END_Attrib
1 1 @F @F @F @F

@Var @RT(9)cMoveNone @RT(0) @T @F @DT @RT(4)DINT @RT(0) @T @T @BASIC 0 @F
@F @F
@T
@BEG_Attrib
0 @RT(13)cMinMoveIdent @RT(4)None
@END_Attrib
1 1 @F @F @F @F

@END_Const

@BEG_Export

@BEG_Kind
@FUNCTION_BLOCK @RT(14)FBManualButton @STRUCTURED_TEXT
@RT(0) @RT(0) @RT(0)
@END_Kind

@BEG_Dcl
@RT(16)DclTreeContainer
15
@Var @RT(7)bButton @RT(0) @T @F @DT @RT(4)BOOL @RT(0) @T @T @BASIC 0 @F
@F @F
@T
@BEG_Attrib
3 @RT(0) @RT(0) @RT(0)
@END_Attrib
1 1 @F @F @F @F

@Var @RT(6)MoveId @RT(0) @T @T @DERIVED 0 @T @T @DT @RT(10)tMoveIdent @RT(0) @T @T @UNKNOWN 0 @F
@F @F
@T
@BEG_Attrib
3 @RT(0) @RT(0) @RT(0)
@END_Attrib
1 1 @F @F @F @F

@Var @RT(7)MoveDir @RT(0) @T @T @DERIVED 0 @T @T @DT @RT(10)tMoveIdent @RT(0) @T @T @UNKNOWN 0 @F
@F @F
@T
@BEG_Attrib
3 @RT(0) @RT(0) @RT(0)
@END_Attrib
1 1 @F @F @F @F

@Var @RT(16)IntermediateCond @RT(0) @T @F @DT @RT(4)DINT @RT(0) @T @T @BASIC 0 @F
@F @F
@T
@BEG_Attrib
3 @RT(0) @RT(0) @RT(0)
@END_Attrib
1 1 @F @F @F @F

@Var @RT(15)sv_bDeviceReady @RT(0) @T @F @DT @RT(4)BOOL @RT(0) @T @T @BASIC 0 @F
@F @F
@T
@BEG_Attrib
3 @RT(0) @RT(0) @RT(0)
@END_Attrib
1 8 @F @F @F @F

@Var @RT(16)sv_OperationMode @RT(0) @T @T @DERIVED 0 @T @T @DT @RT(15)tnOperationMode @RT(0) @T @T @UNKNOWN 0 @F
@F @F
@T
@BEG_Attrib
3 @RT(0) @RT(0) @RT(0)
@END_Attrib
1 8 @F @F @F @F

@Var @RT(11)sv_DeviceId @RT(0) @T @T @DERIVED 0 @T @T @DT @RT(10)tsDeviceId @RT(0) @T @T @UNKNOWN 0 @F
@F @F
@T
@BEG_Attrib
3 @RT(0) @RT(0) @RT(0)
@END_Attrib
1 8 @F @F @F @F

@Var @RT(20)sv_bAutoCalibRunning @RT(0) @T @F @DT @RT(4)BOOL @RT(0) @T @T @BASIC 0 @F
@F @F
@T
@BEG_Attrib
3 @RT(0) @RT(0) @RT(0)
@END_Attrib
1 8 @F @F @F @F

@Var @RT(14)evStartRequest @RT(0) @T @T @DERIVED 0 @T @T @DT @RT(15)tevStartRequest @RT(0) @T @T @UNKNOWN 0 @F
@F @F
@T
@BEG_Attrib
3 @RT(0) @RT(0) @RT(0)
@END_Attrib
1 7 @F @F @F @F

@Var @RT(13)evStopRequest @RT(0) @T @T @DERIVED 0 @T @T @DT @RT(14)tevStopRequest @RT(0) @T @T @UNKNOWN 0 @F
@F @F
@T
@BEG_Attrib
3 @RT(0) @RT(0) @RT(0)
@END_Attrib
1 7 @F @F @F @F

@Var @RT(12)ActiveMoveId @RT(0) @T @T @DERIVED 0 @T @T @DT @RT(10)tMoveIdent @RT(0) @T @T @UNKNOWN 0 @F
@F @F
@T
@BEG_Attrib
3 @RT(0) @RT(0) @RT(0)
@END_Attrib
1 0 @F @F @F @F

@Var @RT(13)ActiveMoveDir @RT(0) @T @T @DERIVED 0 @T @T @DT @RT(10)tMoveIdent @RT(0) @T @T @UNKNOWN 0 @F
@F @F
@T
@BEG_Attrib
3 @RT(0) @RT(0) @RT(0)
@END_Attrib
1 0 @F @F @F @F

@Var @RT(18)evStartRequestData @RT(0) @T @T @DERIVED 0 @T @T @DT @RT(19)tevStartRequestData @RT(0) @T @T @UNKNOWN 0 @F
@F @F
@T
@BEG_Attrib
3 @RT(0) @RT(0) @RT(0)
@END_Attrib
1 0 @F @F @F @F

@Var @RT(17)evStopRequestData @RT(0) @T @T @DERIVED 0 @T @T @DT @RT(18)tevStopRequestData @RT(0) @T @T @UNKNOWN 0 @F
@F @F
@T
@BEG_Attrib
3 @RT(0) @RT(0) @RT(0)
@END_Attrib
1 0 @F @F @F @F

@Var @RT(24)sv_bSequenceInterruption @RT(0) @T @F @DT @RT(4)BOOL @RT(0) @T @T @BASIC 0 @F
@F @F
@T
@BEG_Attrib
3 @RT(0) @RT(29)TRUE: sequence is interrupted @RT(0)
@END_Attrib
1 8 @F @F @F @F

@END_Dcl

@END_Export

@BEG_Body
@TL(48)
(**************************************** WARNING ********************************************
 *** The KEBA Kemro K2 System including software is not intended for safety control tasks! ***
 ***                       For further information see Comment tab!                        ***
 *********************************************************************************************)

IF ((sv_OperationMode >= nHalfAutomatic) AND NOT sv_bSequenceInterruption) OR sv_bAutoCalibRunning THEN
   //do not react on manual buttons in half or fullauto mode or during active autocalibration
   //if sequence is interrupted, some movements are allowed
   RETURN;
END_IF;

IF MoveId > 0 AND
   MoveDir > 0 THEN

   // only start movement if butten is not currently running another movement
   IF bButton AND sv_bDeviceReady AND
      ActiveMoveDir = cMoveNone AND
      ActiveMoveId = cMoveNone THEN

      // remember active movement in case button is used for 2 different MoveID/MoveDir
      // so pressing the second button can not cause any problems
      ActiveMoveDir := MoveDir;
      ActiveMoveId := MoveId;

      // send start request
      evStartRequestData.DeviceId := sv_DeviceId;
      evStartRequestData.MoveDir := MoveDir;
      evStartRequestData.MoveId := MoveId;
      evStartRequestData.IntermediateCond := IntermediateCond;
      SET_EVENT(evStartRequest, evStartRequestData);

   END_IF;

   IF NOT bButton AND
      MoveDir = ActiveMoveDir AND
      MoveId  = ActiveMoveId THEN

      //stop Movement
      evStopRequestData.DeviceId := sv_DeviceId;
      evStopRequestData.MoveDir := ActiveMoveDir;
      evStopRequestData.MoveId := ActiveMoveId;
      SET_EVENT(evStopRequest, evStopRequestData);

      ActiveMoveDir := cMoveNone;
      ActiveMoveId := cMoveNone;
   END_IF;
END_IF;

@END_Body

@END_Contents

(* ---- FBManualButtonKeep.pu ---- *)
(*
Send evStartRequest and evStopRequest events to start a manual movement with a button.

bButton should represent the actual state of the button
(pressed/released)

In half or full auto mode this block will not
react to button press/release
and thus will not send evStartRequest or evStopRequest events.

This FB has a sticky behavior.
On first button press start the movement.
On second button press stop the movement.

Attention:
The same instance of FBManualButtonKeep can not be used for 2 different buttons!
*)

IMPORT_OVER_LISTFILE
 SET_EVENT
, nHalfAutomatic
, tMoveIdent
, tsDeviceId
, tnOperationMode
, tevStartRequest
, tevStopRequest
, tevStartRequestData
, tevStopRequestData

END_IMPORT

FUNCTION_BLOCK FBManualButtonKeep #DUMMY_EDIT_BLOCK

VAR_INPUT
 bButton : BOOL;
 MoveId : tMoveIdent;
 MoveDir : tMoveIdent;
 IntermediateCond : DINT;
END_VAR

SYSTEM_VAR
 sv_DeviceId : tsDeviceId;
 sv_bDeviceReady : BOOL;
 sv_OperationMode : tnOperationMode;
 sv_bAutoCalibRunning : BOOL;
 sv_bSequenceInterruption : BOOL (* TRUE: sequence is interrupted *);
END_VAR

SYSTEM_OBJECT
 evStartRequest : tevStartRequest;
 evStopRequest : tevStopRequest;
END_OBJECT

VAR
 ActiveMoveId : tMoveIdent;
 ActiveMoveDir : tMoveIdent;
 evStartRequestData : tevStartRequestData;
 evStopRequestData : tevStopRequestData;
END_VAR
#BEGIN_EDIT_BLOCK
(**************************************** WARNING ********************************************
 *** The KEBA Kemro K2 System including software is not intended for safety control tasks! ***
 ***                       For further information see Comment tab!                        ***
 *********************************************************************************************)

IF ((sv_OperationMode >= nHalfAutomatic) AND NOT sv_bSequenceInterruption) OR sv_bAutoCalibRunning THEN
   //do not react on manual buttons in half or fullauto mode or during active autocalibration
   //if sequence is interrupted, some movements are allowed
   RETURN;
END_IF;

IF MoveId > 0 AND MoveDir > 0 THEN

   IF bButton THEN
      IF sv_bDeviceReady THEN
         //start Movement
         ActiveMoveDir := MoveDir;
         ActiveMoveId := MoveId;

         // send start request
         evStartRequestData.DeviceId := sv_DeviceId;
         evStartRequestData.MoveDir := MoveDir;
         evStartRequestData.MoveId := MoveId;
         evStartRequestData.IntermediateCond := IntermediateCond;
         SET_EVENT(evStartRequest, evStartRequestData);
      ELSE
         IF MoveDir = ActiveMoveDir AND MoveId = ActiveMoveId THEN
            //stop Movement
            evStopRequestData.DeviceId := sv_DeviceId;
            evStopRequestData.MoveDir := MoveDir;
            evStopRequestData.MoveId := MoveId;
            SET_EVENT(evStopRequest, evStopRequestData);
         END_IF;
      END_IF;
   END_IF;
END_IF;

;#END_EDIT_BLOCK END_FUNCTION_BLOCK

#END_OF_IEC_PART

@Puma @IecEditor 6 114 @Pou 25
@@@BEG_Comment@@@
Send evStartRequest and evStopRequest events to start a manual movement with a button.

bButton should represent the actual state of the button
(pressed/released)

In half or full auto mode this block will not
react to button press/release
and thus will not send evStartRequest or evStopRequest events.

This FB has a sticky behavior.
On first button press start the movement.
On second button press stop the movement.

Attention:
The same instance of FBManualButtonKeep can not be used for 2 different buttons!
@@@END_Comment@@@

@BEG_Contents

@BEG_Func
@RT(17)FuncTreeContainer
1
@Var @RT(9)SET_EVENT @RT(0) @T @T @DERIVED 0 @F @RT(23)KEBA_STANDARD_PROCEDURE @F
@T
@BEG_Attrib
0 @RT(0) @RT(0)
@END_Attrib
1 1 @F @F @F @F

@END_Func

@BEG_Const
@RT(18)ConstTreeContainer
1
@Var @RT(14)nHalfAutomatic @RT(0) @T @T @DERIVED 0 @F @RT(15)tnOperationMode @F
@T
@BEG_Attrib
0 @RT(1)2 @RT(34)confirmation every cycle necessary
@END_Attrib
1 1 @F @F @F @F

@END_Const

@BEG_Export

@BEG_Kind
@FUNCTION_BLOCK @RT(18)FBManualButtonKeep @STRUCTURED_TEXT
@RT(0) @RT(0) @RT(0)
@END_Kind

@BEG_Dcl
@RT(16)DclTreeContainer
15
@Var @RT(7)bButton @RT(0) @T @F @DT @RT(4)BOOL @RT(0) @T @T @BASIC 0 @F
@F @F
@T
@BEG_Attrib
3 @RT(0) @RT(0) @RT(0)
@END_Attrib
1 1 @F @F @F @F

@Var @RT(6)MoveId @RT(0) @T @T @DERIVED 0 @T @T @DT @RT(10)tMoveIdent @RT(0) @T @T @UNKNOWN 0 @F
@F @F
@T
@BEG_Attrib
3 @RT(0) @RT(0) @RT(0)
@END_Attrib
1 1 @F @F @F @F

@Var @RT(7)MoveDir @RT(0) @T @T @DERIVED 0 @T @T @DT @RT(10)tMoveIdent @RT(0) @T @T @UNKNOWN 0 @F
@F @F
@T
@BEG_Attrib
3 @RT(0) @RT(0) @RT(0)
@END_Attrib
1 1 @F @F @F @F

@Var @RT(16)IntermediateCond @RT(0) @T @F @DT @RT(4)DINT @RT(0) @T @T @BASIC 0 @F
@F @F
@T
@BEG_Attrib
3 @RT(0) @RT(0) @RT(0)
@END_Attrib
1 1 @F @F @F @F

@Var @RT(11)sv_DeviceId @RT(0) @T @T @DERIVED 0 @T @T @DT @RT(10)tsDeviceId @RT(0) @T @T @UNKNOWN 0 @F
@F @F
@T
@BEG_Attrib
3 @RT(0) @RT(0) @RT(0)
@END_Attrib
1 8 @F @F @F @F

@Var @RT(15)sv_bDeviceReady @RT(0) @T @F @DT @RT(4)BOOL @RT(0) @T @T @BASIC 0 @F
@F @F
@T
@BEG_Attrib
3 @RT(0) @RT(0) @RT(0)
@END_Attrib
1 8 @F @F @F @F

@Var @RT(16)sv_OperationMode @RT(0) @T @T @DERIVED 0 @T @T @DT @RT(15)tnOperationMode @RT(0) @T @T @UNKNOWN 0 @F
@F @F
@T
@BEG_Attrib
3 @RT(0) @RT(0) @RT(0)
@END_Attrib
1 8 @F @F @F @F

@Var @RT(20)sv_bAutoCalibRunning @RT(0) @T @F @DT @RT(4)BOOL @RT(0) @T @T @BASIC 0 @F
@F @F
@T
@BEG_Attrib
3 @RT(0) @RT(0) @RT(0)
@END_Attrib
1 8 @F @F @F @F

@Var @RT(14)evStartRequest @RT(0) @T @T @DERIVED 0 @T @T @DT @RT(15)tevStartRequest @RT(0) @T @T @UNKNOWN 0 @F
@F @F
@T
@BEG_Attrib
3 @RT(0) @RT(0) @RT(0)
@END_Attrib
1 7 @F @F @F @F

@Var @RT(13)evStopRequest @RT(0) @T @T @DERIVED 0 @T @T @DT @RT(14)tevStopRequest @RT(0) @T @T @UNKNOWN 0 @F
@F @F
@T
@BEG_Attrib
3 @RT(0) @RT(0) @RT(0)
@END_Attrib
1 7 @F @F @F @F

@Var @RT(12)ActiveMoveId @RT(0) @T @T @DERIVED 0 @T @T @DT @RT(10)tMoveIdent @RT(0) @T @T @UNKNOWN 0 @F
@F @F
@T
@BEG_Attrib
3 @RT(0) @RT(0) @RT(0)
@END_Attrib
1 0 @F @F @F @F

@Var @RT(13)ActiveMoveDir @RT(0) @T @T @DERIVED 0 @T @T @DT @RT(10)tMoveIdent @RT(0) @T @T @UNKNOWN 0 @F
@F @F
@T
@BEG_Attrib
3 @RT(0) @RT(0) @RT(0)
@END_Attrib
1 0 @F @F @F @F

@Var @RT(18)evStartRequestData @RT(0) @T @T @DERIVED 0 @T @T @DT @RT(19)tevStartRequestData @RT(0) @T @T @UNKNOWN 0 @F
@F @F
@T
@BEG_Attrib
3 @RT(0) @RT(0) @RT(0)
@END_Attrib
1 0 @F @F @F @F

@Var @RT(17)evStopRequestData @RT(0) @T @T @DERIVED 0 @T @T @DT @RT(18)tevStopRequestData @RT(0) @T @T @UNKNOWN 0 @F
@F @F
@T
@BEG_Attrib
3 @RT(0) @RT(0) @RT(0)
@END_Attrib
1 0 @F @F @F @F

@Var @RT(24)sv_bSequenceInterruption @RT(0) @T @F @DT @RT(4)BOOL @RT(0) @T @T @BASIC 0 @F
@F @F
@T
@BEG_Attrib
3 @RT(0) @RT(29)TRUE: sequence is interrupted @RT(0)
@END_Attrib
1 8 @F @F @F @F

@END_Dcl

@END_Export

@BEG_Body
@TL(37)
(**************************************** WARNING ********************************************
 *** The KEBA Kemro K2 System including software is not intended for safety control tasks! ***
 ***                       For further information see Comment tab!                        ***
 *********************************************************************************************)

IF ((sv_OperationMode >= nHalfAutomatic) AND NOT sv_bSequenceInterruption) OR sv_bAutoCalibRunning THEN
   //do not react on manual buttons in half or fullauto mode or during active autocalibration
   //if sequence is interrupted, some movements are allowed
   RETURN;
END_IF;

IF MoveId > 0 AND MoveDir > 0 THEN

   IF bButton THEN
      IF sv_bDeviceReady THEN
         //start Movement
         ActiveMoveDir := MoveDir;
         ActiveMoveId := MoveId;

         // send start request
         evStartRequestData.DeviceId := sv_DeviceId;
         evStartRequestData.MoveDir := MoveDir;
         evStartRequestData.MoveId := MoveId;
         evStartRequestData.IntermediateCond := IntermediateCond;
         SET_EVENT(evStartRequest, evStartRequestData);
      ELSE
         IF MoveDir = ActiveMoveDir AND MoveId = ActiveMoveId THEN
            //stop Movement
            evStopRequestData.DeviceId := sv_DeviceId;
            evStopRequestData.MoveDir := MoveDir;
            evStopRequestData.MoveId := MoveId;
            SET_EVENT(evStopRequest, evStopRequestData);
         END_IF;
      END_IF;
   END_IF;
END_IF;

@END_Body

@END_Contents

(* ---- FBOpModeAutoLock.pu ---- *)
(*
@h    ! WARNING !
@h    The Kemro K2 system (including software) only meets category B according to EN 954-1,
@h    thus it is not intended for usage in safety-relevant control applications in the field
@h    of personal safety (e.g. emergency stop).
@h    To implement potentially necessary safety-relevant control tasks, always use additional
@h    external safety devices that are intended for the particular purpose, and meet the necessary
@h    functional safety.
@h    For further information see EN 954-1 (EN ISO 13849-1) and/or the K2-x00 user manual, chapter
@h    "CE conformity, directives and standards".

FB to lock and unlock half- and fullautomatic mode.
If IMM is already in automatic mode, no locking takes place, the output flag "bLocked" stays false.
*)

IMPORT_OVER_LISTFILE
 tnOperationMode
, tsLockOperationModeAuto
, FBResourceLock
, KSYS_Status

END_IMPORT

FUNCTION_BLOCK FBOpModeAutoLock #DUMMY_EDIT_BLOCK

VAR_INPUT
 Execute : BOOL;
 bLock : BOOL;
END_VAR

VAR_OUTPUT
 Done : BOOL;
 bLocked : BOOL;
END_VAR

SYSTEM_VAR
 sv_OperationMode : tnOperationMode;
 sv_LockOperationModeAuto : tsLockOperationModeAuto;
END_VAR

VAR
 iStep : DINT;
 bExecuteOld : BOOL;
 bLockIntern : BOOL;
 fbResourceLock : FBResourceLock;
 pDemandedOpMode : REFTO tnOperationMode;
 s : KSYS_Status;
END_VAR
#BEGIN_EDIT_BLOCK
IF (iStep = 0) THEN
    IF (pDemandedOpMode = EMPTY) THEN
        pDemandedOpMode := GET_SYNC_REFTO("OperationMode1.sv_DemandedOperationMode", T#0s, s);
    END_IF;
    IF (Execute AND (NOT bExecuteOld)) THEN
        bLockIntern := bLock;
        Done := FALSE;
        iStep := 10;
    END_IF;
    bExecuteOld := Execute;
END_IF;

IF (iStep = 10) THEN
    IF (bLockIntern = bLocked) THEN
       iStep := 100;
    ELSE
        IF (sv_OperationMode <= nManual) THEN
            fbResourceLock(Execute := FALSE);
            iStep := 20;
        ELSE
            // lock not possible because already in automatic mode
            iStep := 100;
        END_IF;
    END_IF;
END_IF;

IF (iStep = 20) THEN
    fbResourceLock(TRUE, TRUE, @sv_LockOperationModeAuto.sResourceLock);
    IF (fbResourceLock.Done) THEN
        IF (fbResourceLock.bLocked) THEN
           iStep := 30;
        ELSE
           iStep := 100;
        END_IF;
    END_IF;
END_IF;

IF (iStep = 30) THEN
    IF (bLockIntern) THEN
        bLocked := TRUE;
        sv_LockOperationModeAuto.iLockCounter := sv_LockOperationModeAuto.iLockCounter + 1;
        IF ((sv_OperationMode > nManual) OR (pDemandedOpMode^ > nManual)) THEN
            // already in automatic mode or automatic mode requested
            bLocked := FALSE;
            sv_LockOperationModeAuto.iLockCounter := sv_LockOperationModeAuto.iLockCounter - 1;
        END_IF;
    ELSE
        bLocked := FALSE;
        sv_LockOperationModeAuto.iLockCounter := sv_LockOperationModeAuto.iLockCounter - 1;
    END_IF;

    fbResourceLock(bLock := FALSE);
    iStep := 100;
END_IF;

IF (iStep = 100) THEN
    iStep := 0;
    Done := TRUE;
END_IF;

;#END_EDIT_BLOCK END_FUNCTION_BLOCK

#END_OF_IEC_PART

@Puma @IecEditor 6 165 @Pou 25
@@@BEG_Comment@@@
@h    ! WARNING !
@h    The Kemro K2 system (including software) only meets category B according to EN 954-1,
@h    thus it is not intended for usage in safety-relevant control applications in the field
@h    of personal safety (e.g. emergency stop).
@h    To implement potentially necessary safety-relevant control tasks, always use additional
@h    external safety devices that are intended for the particular purpose, and meet the necessary
@h    functional safety.
@h    For further information see EN 954-1 (EN ISO 13849-1) and/or the K2-x00 user manual, chapter
@h    "CE conformity, directives and standards".

FB to lock and unlock half- and fullautomatic mode.
If IMM is already in automatic mode, no locking takes place, the output flag "bLocked" stays false.
@@@END_Comment@@@

@BEG_Contents

@BEG_Func
@RT(17)FuncTreeContainer
0
@END_Func

@BEG_Const
@RT(18)ConstTreeContainer
0
@END_Const

@BEG_Export

@BEG_Kind
@FUNCTION_BLOCK @RT(16)FBOpModeAutoLock @STRUCTURED_TEXT
@RT(0) @RT(0) @RT(0)
@END_Kind

@BEG_Dcl
@RT(16)DclTreeContainer
12
@Var @RT(16)sv_OperationMode @RT(0) @T @T @DERIVED 0 @T @T @DT @RT(15)tnOperationMode @RT(0) @T @T @UNKNOWN 0 @F
@F @F
@T
@BEG_Attrib
3 @RT(0) @RT(0) @RT(0)
@END_Attrib
1 8 @F @F @F @F

@Var @RT(24)sv_LockOperationModeAuto @RT(0) @T @T @DERIVED 0 @T @T @DT @RT(23)tsLockOperationModeAuto @RT(0) @T @T @UNKNOWN 0 @F
@F @F
@T
@BEG_Attrib
3 @RT(0) @RT(0) @RT(0)
@END_Attrib
1 8 @F @F @F @F

@Var @RT(7)Execute @RT(0) @T @F @DT @RT(4)BOOL @RT(0) @T @T @BASIC 0 @F
@F @F
@T
@BEG_Attrib
3 @RT(0) @RT(0) @RT(0)
@END_Attrib
1 1 @F @F @F @F

@Var @RT(5)bLock @RT(0) @T @F @DT @RT(4)BOOL @RT(0) @T @T @BASIC 0 @F
@F @F
@T
@BEG_Attrib
3 @RT(0) @RT(0) @RT(0)
@END_Attrib
1 1 @F @F @F @F

@Var @RT(4)Done @RT(0) @T @F @DT @RT(4)BOOL @RT(0) @T @T @BASIC 0 @F
@F @F
@T
@BEG_Attrib
3 @RT(0) @RT(0) @RT(0)
@END_Attrib
1 3 @F @F @F @F

@Var @RT(7)bLocked @RT(0) @T @F @DT @RT(4)BOOL @RT(0) @T @T @BASIC 0 @F
@F @F
@T
@BEG_Attrib
3 @RT(0) @RT(0) @RT(0)
@END_Attrib
1 3 @F @F @F @F

@Var @RT(5)iStep @RT(0) @T @F @DT @RT(4)DINT @RT(0) @T @T @BASIC 0 @F
@F @F
@T
@BEG_Attrib
3 @RT(0) @RT(0) @RT(0)
@END_Attrib
1 0 @F @F @F @F

@Var @RT(11)bExecuteOld @RT(0) @T @F @DT @RT(4)BOOL @RT(0) @T @T @BASIC 0 @F
@F @F
@T
@BEG_Attrib
3 @RT(0) @RT(0) @RT(0)
@END_Attrib
1 0 @F @F @F @F

@Var @RT(11)bLockIntern @RT(0) @T @F @DT @RT(4)BOOL @RT(0) @T @T @BASIC 0 @F
@F @F
@T
@BEG_Attrib
3 @RT(0) @RT(0) @RT(0)
@END_Attrib
1 0 @F @F @F @F

@Var @RT(14)fbResourceLock @RT(0) @T @T @DERIVED 0 @T @T @DT @RT(14)FBResourceLock @RT(0) @T @T @UNKNOWN 0 @F
@F @F
@T
@BEG_Attrib
3 @RT(0) @RT(0) @RT(0)
@END_Attrib
1 0 @F @F @F @F

@Var @RT(15)pDemandedOpMode @RT(0) @T @T @REFTO 0 @F @DERIVED 0 @T @T @DT @RT(15)tnOperationMode @RT(0) @T @T @UNKNOWN 0 @F
@F @F
@T
@BEG_Attrib
3 @RT(0) @RT(0) @RT(0)
@END_Attrib
1 0 @F @F @F @F

@Var @RT(1)s @RT(0) @T @T @DERIVED 0 @T @T @DT @RT(11)KSYS_Status @RT(0) @T @T @UNKNOWN 0 @F
@F @F
@T
@BEG_Attrib
3 @RT(0) @RT(0) @RT(0)
@END_Attrib
1 0 @F @F @F @F

@END_Dcl

@END_Export

@BEG_Body
@TL(61)
IF (iStep = 0) THEN
    IF (pDemandedOpMode = EMPTY) THEN
        pDemandedOpMode := GET_SYNC_REFTO("OperationMode1.sv_DemandedOperationMode", T#0s, s);
    END_IF;
    IF (Execute AND (NOT bExecuteOld)) THEN
        bLockIntern := bLock;
        Done := FALSE;
        iStep := 10;
    END_IF;
    bExecuteOld := Execute;
END_IF;

IF (iStep = 10) THEN
    IF (bLockIntern = bLocked) THEN
       iStep := 100;
    ELSE
        IF (sv_OperationMode <= nManual) THEN
            fbResourceLock(Execute := FALSE);
            iStep := 20;
        ELSE
            // lock not possible because already in automatic mode
            iStep := 100;
        END_IF;
    END_IF;
END_IF;

IF (iStep = 20) THEN
    fbResourceLock(TRUE, TRUE, @sv_LockOperationModeAuto.sResourceLock);
    IF (fbResourceLock.Done) THEN
        IF (fbResourceLock.bLocked) THEN
           iStep := 30;
        ELSE
           iStep := 100;
        END_IF;
    END_IF;
END_IF;

IF (iStep = 30) THEN
    IF (bLockIntern) THEN
        bLocked := TRUE;
        sv_LockOperationModeAuto.iLockCounter := sv_LockOperationModeAuto.iLockCounter + 1;
        IF ((sv_OperationMode > nManual) OR (pDemandedOpMode^ > nManual)) THEN
            // already in automatic mode or automatic mode requested
            bLocked := FALSE;
            sv_LockOperationModeAuto.iLockCounter := sv_LockOperationModeAuto.iLockCounter - 1;
        END_IF;
    ELSE
        bLocked := FALSE;
        sv_LockOperationModeAuto.iLockCounter := sv_LockOperationModeAuto.iLockCounter - 1;
    END_IF;

    fbResourceLock(bLock := FALSE);
    iStep := 100;
END_IF;

IF (iStep = 100) THEN
    iStep := 0;
    Done := TRUE;
END_IF;

@END_Body

@END_Contents

(* ---- FBOpModeHalfAndAutoEntered.pu ---- *)
(*
@h    ! WARNING !
@h    The Kemro K2 system (including software) only meets category B according to EN 954-1,
@h    thus it is not intended for usage in safety-relevant control applications in the field
@h    of personal safety (e.g. emergency stop).
@h    To implement potentially necessary safety-relevant control tasks, always use additional
@h    external safety devices that are intended for the particular purpose, and meet the necessary
@h    functional safety.
@h    For further information see EN 954-1 (EN ISO 13849-1) and/or the K2-x00 user manual, chapter
@h    "CE conformity, directives and standards".

output Q is TRUE if operationmode changes from setup- or manualmode to full- or halfauto mode
*)

IMPORT_OVER_LISTFILE
 R_TRIG
, tnOperationMode

END_IMPORT

FUNCTION_BLOCK FBOpModeHalfAndAutoEntered #DUMMY_EDIT_BLOCK

VAR_INPUT
 iOperationMode : tnOperationMode;
END_VAR

VAR_OUTPUT
 Q : BOOL;
END_VAR

VAR
 fbRTrig : R_TRIG;
END_VAR
#BEGIN_EDIT_BLOCK
(**************************************** WARNING ********************************************
 *** The KEBA Kemro K2 System including software is not intended for safety control tasks! ***
 ***                       For further information see Comment tab!                        ***
 *********************************************************************************************)

fbRTrig(CLK := iOperationMode > nManual);
Q := fbRTrig.Q;

;#END_EDIT_BLOCK END_FUNCTION_BLOCK

#END_OF_IEC_PART

@Puma @IecEditor 6 150 @Pou 25
@@@BEG_Comment@@@
@h    ! WARNING !
@h    The Kemro K2 system (including software) only meets category B according to EN 954-1,
@h    thus it is not intended for usage in safety-relevant control applications in the field
@h    of personal safety (e.g. emergency stop).
@h    To implement potentially necessary safety-relevant control tasks, always use additional
@h    external safety devices that are intended for the particular purpose, and meet the necessary
@h    functional safety.
@h    For further information see EN 954-1 (EN ISO 13849-1) and/or the K2-x00 user manual, chapter
@h    "CE conformity, directives and standards".

output Q is TRUE if operationmode changes from setup- or manualmode to full- or halfauto mode
@@@END_Comment@@@

@BEG_Contents

@BEG_Func
@RT(17)FuncTreeContainer
0
@END_Func

@BEG_Const
@RT(18)ConstTreeContainer
0
@END_Const

@BEG_Export

@BEG_Kind
@FUNCTION_BLOCK @RT(26)FBOpModeHalfAndAutoEntered @STRUCTURED_TEXT
@RT(0) @RT(0) @RT(0)
@END_Kind

@BEG_Dcl
@RT(16)DclTreeContainer
3
@Var @RT(7)fbRTrig @RT(0) @T @T @DERIVED 0 @F @RT(6)R_TRIG @F
@T
@BEG_Attrib
3 @RT(0) @RT(0) @RT(0)
@END_Attrib
1 0 @F @F @F @F

@Var @RT(14)iOperationMode @RT(0) @T @T @DERIVED 0 @F @RT(15)tnOperationMode @F
@T
@BEG_Attrib
3 @RT(0) @RT(0) @RT(0)
@END_Attrib
1 1 @F @F @F @F

@Var @RT(1)Q @RT(0) @T @F @DT @RT(4)BOOL @RT(0) @T @T @BASIC 0 @F
@F @F
@T
@BEG_Attrib
3 @RT(0) @RT(0) @RT(0)
@END_Attrib
1 3 @F @F @F @F

@END_Dcl

@END_Export

@BEG_Body
@TL(8)
(**************************************** WARNING ********************************************
 *** The KEBA Kemro K2 System including software is not intended for safety control tasks! ***
 ***                       For further information see Comment tab!                        ***
 *********************************************************************************************)

fbRTrig(CLK := iOperationMode > nManual);
Q := fbRTrig.Q;

@END_Body

@END_Contents

(* ---- FBOpModeHalfAndAutoLeft.pu ---- *)
(*
@h    ! WARNING !
@h    The Kemro K2 system (including software) only meets category B according to EN 954-1,
@h    thus it is not intended for usage in safety-relevant control applications in the field
@h    of personal safety (e.g. emergency stop).
@h    To implement potentially necessary safety-relevant control tasks, always use additional
@h    external safety devices that are intended for the particular purpose, and meet the necessary
@h    functional safety.
@h    For further information see EN 954-1 (EN ISO 13849-1) and/or the K2-x00 user manual, chapter
@h    "CE conformity, directives and standards".

output Q is TRUE if operationmode changes from full- or halfauto mode to setup- or manualmode
*)

IMPORT_OVER_LISTFILE
 F_TRIG
, tnOperationMode

END_IMPORT

FUNCTION_BLOCK FBOpModeHalfAndAutoLeft #DUMMY_EDIT_BLOCK

VAR_INPUT
 iOperationMode : tnOperationMode;
END_VAR

VAR_OUTPUT
 Q : BOOL;
END_VAR

VAR
 fbFTrig : F_TRIG;
END_VAR
#BEGIN_EDIT_BLOCK
(**************************************** WARNING ********************************************
 *** The KEBA Kemro K2 System including software is not intended for safety control tasks! ***
 ***                       For further information see Comment tab!                        ***
 *********************************************************************************************)

fbFTrig(CLK := iOperationMode > nManual);
Q := fbFTrig.Q;

;#END_EDIT_BLOCK END_FUNCTION_BLOCK

#END_OF_IEC_PART

@Puma @IecEditor 6 150 @Pou 25
@@@BEG_Comment@@@
@h    ! WARNING !
@h    The Kemro K2 system (including software) only meets category B according to EN 954-1,
@h    thus it is not intended for usage in safety-relevant control applications in the field
@h    of personal safety (e.g. emergency stop).
@h    To implement potentially necessary safety-relevant control tasks, always use additional
@h    external safety devices that are intended for the particular purpose, and meet the necessary
@h    functional safety.
@h    For further information see EN 954-1 (EN ISO 13849-1) and/or the K2-x00 user manual, chapter
@h    "CE conformity, directives and standards".

output Q is TRUE if operationmode changes from full- or halfauto mode to setup- or manualmode
@@@END_Comment@@@

@BEG_Contents

@BEG_Func
@RT(17)FuncTreeContainer
0
@END_Func

@BEG_Const
@RT(18)ConstTreeContainer
0
@END_Const

@BEG_Export

@BEG_Kind
@FUNCTION_BLOCK @RT(23)FBOpModeHalfAndAutoLeft @STRUCTURED_TEXT
@RT(0) @RT(0) @RT(0)
@END_Kind

@BEG_Dcl
@RT(16)DclTreeContainer
3
@Var @RT(7)fbFTrig @RT(0) @T @T @DERIVED 0 @F @RT(6)F_TRIG @F
@T
@BEG_Attrib
3 @RT(0) @RT(0) @RT(0)
@END_Attrib
1 0 @F @F @F @F

@Var @RT(14)iOperationMode @RT(0) @T @T @DERIVED 0 @T @T @DT @RT(15)tnOperationMode @RT(0) @T @T @UNKNOWN 0 @F
@F @F
@T
@BEG_Attrib
3 @RT(0) @RT(0) @RT(0)
@END_Attrib
1 1 @F @F @F @F

@Var @RT(1)Q @RT(0) @T @F @DT @RT(4)BOOL @RT(0) @T @T @BASIC 0 @F
@F @F
@T
@BEG_Attrib
3 @RT(0) @RT(0) @RT(0)
@END_Attrib
1 3 @F @F @F @F

@END_Dcl

@END_Export

@BEG_Body
@TL(8)
(**************************************** WARNING ********************************************
 *** The KEBA Kemro K2 System including software is not intended for safety control tasks! ***
 ***                       For further information see Comment tab!                        ***
 *********************************************************************************************)

fbFTrig(CLK := iOperationMode > nManual);
Q := fbFTrig.Q;

@END_Body

@END_Contents

(* ---- FBPeakMeasure.pu ---- *)
(*
Function Block for detecting a minimum/maximum peakvalue of an analog signal.

A rising edge on the bTrigger input starts the measurement.
During measurement the rPeakVal output is always updated with the latest peakvalue.
To reset the FB it must be called with bStop=TRUE. Then rPeakVal is set to zero and the FB is ready for a new peakvalue measurement.
bMinMax selects if the maximum or minimum peakvalue should be detected. (FALSE...max, TRUE...min)
*)

FUNCTION_BLOCK FBPeakMeasure #DUMMY_EDIT_BLOCK

VAR_INPUT
 rActVal : REAL (* Actual value input for peak measurement *);
 bTrigger : BOOL (* Boolean trigger input *);
 bReset : BOOL;
 bMinMax : BOOL (* Minimum/Maximum peak value (FALSE: max, TRUE: min) *);
END_VAR

VAR_OUTPUT
 rPeakVal : REAL (* Peak value output *);
END_VAR

VAR
 bTriggered : BOOL;
END_VAR
#BEGIN_EDIT_BLOCK
IF NOT bReset THEN

   IF bTrigger OR bTriggered THEN
      bTriggered := TRUE;

      IF (NOT bMinMax AND (rActVal > rPeakVal)) OR (bMinMax AND (rActVal < rPeakVal)) THEN
          rPeakVal := rActVal;
      END_IF;
   END_IF;
ELSE
   //not OK for MIN
   //rPeakVal := 0.0;
   rPeakVal := rActVal;
   bTriggered := FALSE;
END_IF;

;#END_EDIT_BLOCK END_FUNCTION_BLOCK

#END_OF_IEC_PART

@Puma @IecEditor 6 80 @Pou 25
@@@BEG_Comment@@@
Function Block for detecting a minimum/maximum peakvalue of an analog signal.

A rising edge on the bTrigger input starts the measurement.
During measurement the rPeakVal output is always updated with the latest peakvalue.
To reset the FB it must be called with bStop=TRUE. Then rPeakVal is set to zero and the FB is ready for a new peakvalue measurement.
bMinMax selects if the maximum or minimum peakvalue should be detected. (FALSE...max, TRUE...min)
@@@END_Comment@@@

@BEG_Contents

@BEG_Func
@RT(17)FuncTreeContainer
0
@END_Func

@BEG_Const
@RT(18)ConstTreeContainer
0
@END_Const

@BEG_Export

@BEG_Kind
@FUNCTION_BLOCK @RT(13)FBPeakMeasure @STRUCTURED_TEXT
@RT(0) @RT(0) @RT(0)
@END_Kind

@BEG_Dcl
@RT(16)DclTreeContainer
6
@Var @RT(7)rActVal @RT(0) @T @F @DT @RT(4)REAL @RT(0) @T @T @BASIC 0 @F
@F @F
@T
@BEG_Attrib
3 @RT(0) @RT(39)Actual value input for peak measurement @RT(0)
@END_Attrib
1 1 @F @F @F @F

@Var @RT(8)bTrigger @RT(0) @T @F @DT @RT(4)BOOL @RT(0) @T @T @BASIC 0 @F
@F @F
@T
@BEG_Attrib
3 @RT(0) @RT(21)Boolean trigger input @RT(0)
@END_Attrib
1 1 @F @F @F @F

@Var @RT(6)bReset @RT(0) @T @F @DT @RT(4)BOOL @RT(0) @T @T @BASIC 0 @F
@F @F
@T
@BEG_Attrib
3 @RT(0) @RT(0) @RT(0)
@END_Attrib
1 1 @F @F @F @F

@Var @RT(7)bMinMax @RT(0) @T @F @DT @RT(4)BOOL @RT(0) @T @T @BASIC 0 @F
@F @F
@T
@BEG_Attrib
3 @RT(0) @RT(50)Minimum/Maximum peak value (FALSE: max, TRUE: min) @RT(0)
@END_Attrib
1 1 @F @F @F @F

@Var @RT(8)rPeakVal @RT(0) @T @F @DT @RT(4)REAL @RT(0) @T @T @BASIC 0 @F
@F @F
@T
@BEG_Attrib
3 @RT(0) @RT(17)Peak value output @RT(0)
@END_Attrib
1 3 @F @F @F @F

@Var @RT(10)bTriggered @RT(0) @T @F @DT @RT(4)BOOL @RT(0) @T @T @BASIC 0 @F
@F @F
@T
@BEG_Attrib
3 @RT(0) @RT(0) @RT(0)
@END_Attrib
1 0 @F @F @F @F

@END_Dcl

@END_Export

@BEG_Body
@TL(16)
IF NOT bReset THEN

   IF bTrigger OR bTriggered THEN
      bTriggered := TRUE;

      IF (NOT bMinMax AND (rActVal > rPeakVal)) OR (bMinMax AND (rActVal < rPeakVal)) THEN
          rPeakVal := rActVal;
      END_IF;
   END_IF;
ELSE
   //not OK for MIN
   //rPeakVal := 0.0;
   rPeakVal := rActVal;
   bTriggered := FALSE;
END_IF;

@END_Body

@END_Contents

(* ---- FBResourceLock.pu ---- *)
IMPORT_OVER_LISTFILE
 GET_RUNTIME
, tpsResourceLock

END_IMPORT

FUNCTION_BLOCK FBResourceLock #DUMMY_EDIT_BLOCK

VAR_INPUT
 Execute : BOOL;
 bLock : BOOL;
 pResourceLock : tpsResourceLock;
END_VAR

VAR_OUTPUT
 bLocked : BOOL;
 Done : BOOL;
END_VAR

VAR
 pResourceLockIntern : tpsResourceLock;
 t : TIME;
 iStep : DINT;
 iTmpRequestId : DWORD;
 oldExe : BOOL;
 bLockCntOld : UDINT;
END_VAR
#BEGIN_EDIT_BLOCK
IF (iStep = 0) THEN
    IF (Execute AND (NOT oldExe)) THEN
        iStep := 5;
        pResourceLockIntern := pResourceLock;    // copy reference because of  IEC Generate bug
    END_IF;
END_IF;

oldExe := Execute;

IF (iStep = 5) THEN
    bLocked := FALSE;
    IF (bLock) THEN
      Done := FALSE;
      IF (pResourceLockIntern^.iLocked MOD 2 = 1) THEN
         iStep := 0;
         Done := TRUE;  // no way to get resource, do not even try
      ELSE
         t := GET_RUNTIME(); // getruntime is guaranteed to return a different value each call (see CIkbTypSystem::IecGetRunTime)
         iTmpRequestId := LINT_TO_DWORD(TIME_TO_LINT(t)); // use only lower 31 bits
         iTmpRequestId := iTmpRequestId AND 16#0FFFFFFF;  // highest 4 bits are reserved: bit 31 for IEC, bit 30 for HmiServer, rest for future use
         iTmpRequestId := iTmpRequestId OR 16#80000000;  // set bit 31, request id is never 0

         // iTmpRequestId is guaranteed to be unique for 2^28 µs ~ 270 sec ~ 5 min
         // this is sufficient because unique id is only necessary during race-condition:
         // start of request until response
         bLockCntOld := pResourceLockIntern^.iLocked;
         pResourceLockIntern^.iRequest := iTmpRequestId;
         iStep := 10;
      END_IF;
    ELSE
        iStep := 0;
        Done := TRUE;
    END_IF;
END_IF;

IF (iStep = 10) THEN
     IF (iTmpRequestId = pResourceLockIntern^.iResponse) THEN
         bLocked := TRUE;  // we have won the race
         iStep := 20;
     ELSIF (bLockCntOld <> pResourceLockIntern^.iLocked) THEN // we have lost the race, another client got the lock
         iStep := 0;
         Done := TRUE;
     END_IF;
END_IF;

IF (iStep = 20) THEN
    IF (NOT bLock) THEN
          bLocked := FALSE;
          pResourceLockIntern^.iResponse := 0;
          iStep := 0;
    ELSE
        Done := TRUE;
    END_IF;
END_IF;

;#END_EDIT_BLOCK END_FUNCTION_BLOCK

#END_OF_IEC_PART

@Puma @IecEditor 6 159 @Pou 25
@@@BEG_Comment@@@

@@@END_Comment@@@

@BEG_Contents

@BEG_Func
@RT(17)FuncTreeContainer
1
@Var @RT(11)GET_RUNTIME @RT(0) @T @T @DERIVED 0 @F @RT(22)KEBA_STANDARD_FUNCTION @F
@T
@BEG_Attrib
0 @RT(0) @RT(0)
@END_Attrib
1 1 @F @F @F @F

@END_Func

@BEG_Const
@RT(18)ConstTreeContainer
0
@END_Const

@BEG_Export

@BEG_Kind
@FUNCTION_BLOCK @RT(14)FBResourceLock @STRUCTURED_TEXT
@RT(0) @RT(0) @RT(0)
@END_Kind

@BEG_Dcl
@RT(16)DclTreeContainer
11
@Var @RT(7)Execute @RT(0) @T @F @DT @RT(4)BOOL @RT(0) @T @T @BASIC 0 @F
@F @F
@T
@BEG_Attrib
3 @RT(0) @RT(0) @RT(0)
@END_Attrib
1 1 @F @F @F @F

@Var @RT(5)bLock @RT(0) @T @F @DT @RT(4)BOOL @RT(0) @T @T @BASIC 0 @F
@F @F
@T
@BEG_Attrib
3 @RT(0) @RT(0) @RT(0)
@END_Attrib
1 1 @F @F @F @F

@Var @RT(13)pResourceLock @RT(0) @T @T @DERIVED 0 @T @T @DT @RT(15)tpsResourceLock @RT(0) @T @T @UNKNOWN 0 @F
@F @F
@T
@BEG_Attrib
3 @RT(0) @RT(0) @RT(0)
@END_Attrib
1 1 @F @F @F @F

@Var @RT(19)pResourceLockIntern @RT(0) @T @T @DERIVED 0 @T @T @DT @RT(15)tpsResourceLock @RT(0) @T @T @UNKNOWN 0 @F
@F @F
@T
@BEG_Attrib
3 @RT(0) @RT(0) @RT(0)
@END_Attrib
1 0 @F @F @F @F

@Var @RT(7)bLocked @RT(0) @T @F @DT @RT(4)BOOL @RT(0) @T @T @BASIC 0 @F
@F @F
@T
@BEG_Attrib
3 @RT(0) @RT(0) @RT(0)
@END_Attrib
1 3 @F @F @F @F

@Var @RT(4)Done @RT(0) @T @F @DT @RT(4)BOOL @RT(0) @T @T @BASIC 0 @F
@F @F
@T
@BEG_Attrib
3 @RT(0) @RT(0) @RT(0)
@END_Attrib
1 3 @F @F @F @F

@Var @RT(1)t @RT(0) @T @F @DT @RT(4)TIME @RT(0) @T @T @BASIC 0 @F
@F @F
@T
@BEG_Attrib
3 @RT(0) @RT(0) @RT(0)
@END_Attrib
1 0 @F @F @F @F

@Var @RT(5)iStep @RT(0) @T @F @DT @RT(4)DINT @RT(0) @T @T @BASIC 0 @F
@F @F
@T
@BEG_Attrib
3 @RT(0) @RT(0) @RT(0)
@END_Attrib
1 0 @F @F @F @F

@Var @RT(13)iTmpRequestId @RT(0) @T @F @DT @RT(5)DWORD @RT(0) @T @T @BASIC 0 @F
@F @F
@T
@BEG_Attrib
3 @RT(0) @RT(0) @RT(0)
@END_Attrib
1 0 @F @F @F @F

@Var @RT(6)oldExe @RT(0) @T @F @DT @RT(4)BOOL @RT(0) @T @T @BASIC 0 @F
@F @F
@T
@BEG_Attrib
3 @RT(0) @RT(0) @RT(0)
@END_Attrib
1 0 @F @F @F @F

@Var @RT(11)bLockCntOld @RT(0) @T @F @DT @RT(5)UDINT @RT(0) @T @T @BASIC 0 @F
@F @F
@T
@BEG_Attrib
3 @RT(0) @RT(0) @RT(0)
@END_Attrib
1 0 @F @F @F @F

@END_Dcl

@END_Export

@BEG_Body
@TL(57)
IF (iStep = 0) THEN
    IF (Execute AND (NOT oldExe)) THEN
        iStep := 5;
        pResourceLockIntern := pResourceLock;    // copy reference because of  IEC Generate bug
    END_IF;
END_IF;

oldExe := Execute;

IF (iStep = 5) THEN
    bLocked := FALSE;
    IF (bLock) THEN
      Done := FALSE;
      IF (pResourceLockIntern^.iLocked MOD 2 = 1) THEN
         iStep := 0;
         Done := TRUE;  // no way to get resource, do not even try
      ELSE
         t := GET_RUNTIME(); // getruntime is guaranteed to return a different value each call (see CIkbTypSystem::IecGetRunTime)
         iTmpRequestId := LINT_TO_DWORD(TIME_TO_LINT(t)); // use only lower 31 bits
         iTmpRequestId := iTmpRequestId AND 16#0FFFFFFF;  // highest 4 bits are reserved: bit 31 for IEC, bit 30 for HmiServer, rest for future use
         iTmpRequestId := iTmpRequestId OR 16#80000000;  // set bit 31, request id is never 0

         // iTmpRequestId is guaranteed to be unique for 2^28 µs ~ 270 sec ~ 5 min
         // this is sufficient because unique id is only necessary during race-condition:
         // start of request until response
         bLockCntOld := pResourceLockIntern^.iLocked;
         pResourceLockIntern^.iRequest := iTmpRequestId;
         iStep := 10;
      END_IF;
    ELSE
        iStep := 0;
        Done := TRUE;
    END_IF;
END_IF;

IF (iStep = 10) THEN
     IF (iTmpRequestId = pResourceLockIntern^.iResponse) THEN
         bLocked := TRUE;  // we have won the race
         iStep := 20;
     ELSIF (bLockCntOld <> pResourceLockIntern^.iLocked) THEN // we have lost the race, another client got the lock
         iStep := 0;
         Done := TRUE;
     END_IF;
END_IF;

IF (iStep = 20) THEN
    IF (NOT bLock) THEN
          bLocked := FALSE;
          pResourceLockIntern^.iResponse := 0;
          iStep := 0;
    ELSE
        Done := TRUE;
    END_IF;
END_IF;

@END_Body

@END_Contents

(* ---- FBSetMovementState.pu ---- *)
IMPORT_OVER_LISTFILE
 tevMovementStateData
, tevMovementState
, tMoveIdent
, tnActiveInactive
, tsDeviceId

END_IMPORT

FUNCTION_BLOCK FBSetMovementState #DUMMY_EDIT_BLOCK

VAR_INPUT
 MoveId : tMoveIdent;
 MoveDir : tMoveIdent;
 State : tnActiveInactive;
END_VAR

SYSTEM_VAR
 sv_DeviceId : tsDeviceId;
END_VAR

SYSTEM_OBJECT
 evMovementState : tevMovementState;
END_OBJECT

VAR
 evMovementStateData : tevMovementStateData;
END_VAR
#BEGIN_EDIT_BLOCK
(* Sending evMovementState - used for MovementSymbols in Vis *)
evMovementStateData.DeviceId := sv_DeviceId;
evMovementStateData.MoveId   := MoveId;
evMovementStateData.MoveDir  := MoveDir;
evMovementStateData.State    := State;
SET_EVENT(evMovementState, evMovementStateData);

;#END_EDIT_BLOCK END_FUNCTION_BLOCK

#END_OF_IEC_PART

@Puma @IecEditor 6 10 @Pou 25
@@@BEG_Comment@@@

@@@END_Comment@@@

@BEG_Contents

@BEG_Func
@RT(17)FuncTreeContainer
0
@END_Func

@BEG_Const
@RT(18)ConstTreeContainer
0
@END_Const

@BEG_Export

@BEG_Kind
@FUNCTION_BLOCK @RT(18)FBSetMovementState @STRUCTURED_TEXT
@RT(0) @RT(0) @RT(0)
@END_Kind

@BEG_Dcl
@RT(16)DclTreeContainer
6
@Var @RT(6)MoveId @RT(0) @T @T @DERIVED 0 @F @RT(10)tMoveIdent @F
@T
@BEG_Attrib
3 @RT(0) @RT(0) @RT(0)
@END_Attrib
1 1 @F @F @F @F

@Var @RT(7)MoveDir @RT(0) @T @T @DERIVED 0 @F @RT(10)tMoveIdent @F
@T
@BEG_Attrib
3 @RT(0) @RT(0) @RT(0)
@END_Attrib
1 1 @F @F @F @F

@Var @RT(5)State @RT(0) @T @T @DERIVED 0 @F @RT(16)tnActiveInactive @F
@T
@BEG_Attrib
3 @RT(0) @RT(0) @RT(0)
@END_Attrib
1 1 @F @F @F @F

@Var @RT(19)evMovementStateData @RT(0) @T @T @DERIVED 0 @T @T @DT @RT(20)tevMovementStateData @RT(0) @T @T @UNKNOWN 0 @F
@F @F
@T
@BEG_Attrib
3 @RT(0) @RT(0) @RT(0)
@END_Attrib
1 0 @F @F @F @F

@Var @RT(15)evMovementState @RT(0) @T @T @DERIVED 0 @T @T @DT @RT(16)tevMovementState @RT(0) @T @T @UNKNOWN 0 @F
@F @F
@T
@BEG_Attrib
3 @RT(0) @RT(0) @RT(0)
@END_Attrib
1 7 @F @F @F @F

@Var @RT(11)sv_DeviceId @RT(0) @T @T @DERIVED 0 @T @T @DT @RT(10)tsDeviceId @RT(0) @T @T @UNKNOWN 0 @F
@F @F
@T
@BEG_Attrib
3 @RT(0) @RT(0) @RT(0)
@END_Attrib
1 8 @F @F @F @F

@END_Dcl

@END_Export

@BEG_Body
@TL(7)
(* Sending evMovementState - used for MovementSymbols in Vis *)
evMovementStateData.DeviceId := sv_DeviceId;
evMovementStateData.MoveId   := MoveId;
evMovementStateData.MoveDir  := MoveDir;
evMovementStateData.State    := State;
SET_EVENT(evMovementState, evMovementStateData);

@END_Body

@END_Contents

(* ---- FBSinus.pu ---- *)
(*
@h    ! WARNING !
@h    The Kemro K2 system (including software) only meets category B according to EN 954-1,
@h    thus it is not intended for usage in safety-relevant control applications in the field
@h    of personal safety (e.g. emergency stop).
@h    To implement potentially necessary safety-relevant control tasks, always use additional
@h    external safety devices that are intended for the particular purpose, and meet the necessary
@h    functional safety.
@h    For further information see EN 954-1 (EN ISO 13849-1) and/or the K2-x00 user manual, chapter
@h    "CE conformity, directives and standards".

FB for generating a sinus signal
*)

IMPORT_OVER_LISTFILE
 GET_TASK_INTERVAL
, cApplPlasticsPI

END_IMPORT

FUNCTION_BLOCK FBSinus #DUMMY_EDIT_BLOCK

VAR_INPUT
 rAmplitude : REAL (* amplitude *);
 rFrequency : REAL (* frequency (in Hz) *);
END_VAR

VAR_OUTPUT
 rOut : REAL (* generated sinus value *);
END_VAR

VAR
 rStepWidth : REAL := 0.628319;
 rX : REAL;
 dTaskCycleTime : TIME (* cycle time in ms *);
 bInitDone : BOOL;
 rTaskCycleTime : REAL;
END_VAR
#BEGIN_EDIT_BLOCK
(**************************************** WARNING ********************************************
 *** The KEBA Kemro K2 System including software is not intended for safety control tasks! ***
 ***                       For further information see Comment tab!                        ***
 *********************************************************************************************)

IF NOT bInitDone THEN
   dTaskCycleTime := GET_TASK_INTERVAL();
   rTaskCycleTime := LINT_TO_REAL(TIME_TO_LINT(dTaskCycleTime)) / 1000000.0;   //task cycle time in sec
   bInitDone := TRUE;
END_IF;

rStepWidth := 2.0 * cApplPlasticsPI * rFrequency * rTaskCycleTime;

rOut := rAmplitude * SIN(rX);
rX := rX + rStepWidth;
IF rX > (2.0 * cApplPlasticsPI) THEN
    rX := rX - (2.0 * cApplPlasticsPI);
END_IF;

;#END_EDIT_BLOCK END_FUNCTION_BLOCK

#END_OF_IEC_PART

@Puma @IecEditor 6 113 @Pou 25
@@@BEG_Comment@@@
@h    ! WARNING !
@h    The Kemro K2 system (including software) only meets category B according to EN 954-1,
@h    thus it is not intended for usage in safety-relevant control applications in the field
@h    of personal safety (e.g. emergency stop).
@h    To implement potentially necessary safety-relevant control tasks, always use additional
@h    external safety devices that are intended for the particular purpose, and meet the necessary
@h    functional safety.
@h    For further information see EN 954-1 (EN ISO 13849-1) and/or the K2-x00 user manual, chapter
@h    "CE conformity, directives and standards".

FB for generating a sinus signal
@@@END_Comment@@@

@BEG_Contents

@BEG_Func
@RT(17)FuncTreeContainer
1
@Var @RT(17)GET_TASK_INTERVAL @RT(0) @T @T @DERIVED 0 @F @RT(22)KEBA_STANDARD_FUNCTION @F
@T
@BEG_Attrib
0 @RT(0) @RT(0)
@END_Attrib
1 1 @F @F @F @F

@END_Func

@BEG_Const
@RT(18)ConstTreeContainer
1
@Var @RT(15)cApplPlasticsPI @RT(0) @T @F @DT @RT(4)REAL @RT(0) @T @T @BASIC 0 @F
@F @F
@T
@BEG_Attrib
0 @RT(10)3.14159265 @RT(13)pi=3.14159265
@END_Attrib
1 1 @F @F @F @F

@END_Const

@BEG_Export

@BEG_Kind
@FUNCTION_BLOCK @RT(7)FBSinus @STRUCTURED_TEXT
@RT(0) @RT(0) @RT(0)
@END_Kind

@BEG_Dcl
@RT(16)DclTreeContainer
8
@Var @RT(10)rAmplitude @RT(0) @T @F @DT @RT(4)REAL @RT(0) @T @T @BASIC 0 @F
@F @F
@T
@BEG_Attrib
3 @RT(0) @RT(9)amplitude @RT(0)
@END_Attrib
1 1 @F @F @F @F

@Var @RT(10)rFrequency @RT(0) @T @F @DT @RT(4)REAL @RT(0) @T @T @BASIC 0 @F
@F @F
@T
@BEG_Attrib
3 @RT(0) @RT(17)frequency (in Hz) @RT(0)
@END_Attrib
1 1 @F @F @F @F

@Var @RT(4)rOut @RT(0) @T @F @DT @RT(4)REAL @RT(0) @T @T @BASIC 0 @F
@F @F
@T
@BEG_Attrib
3 @RT(0) @RT(21)generated sinus value @RT(0)
@END_Attrib
1 3 @F @F @F @F

@Var @RT(10)rStepWidth @RT(0) @T @F @DT @RT(4)REAL @RT(0) @T @T @BASIC 0 @F
@F @F
@T
@BEG_Attrib
3 @RT(8)0.628319 @RT(0) @RT(0)
@END_Attrib
1 0 @F @F @F @F

@Var @RT(2)rX @RT(0) @T @F @DT @RT(4)REAL @RT(0) @T @T @BASIC 0 @F
@F @F
@T
@BEG_Attrib
3 @RT(0) @RT(0) @RT(0)
@END_Attrib
1 0 @F @F @F @F

@Var @RT(14)dTaskCycleTime @RT(0) @T @F @DT @RT(4)TIME @RT(0) @T @T @BASIC 0 @F
@F @F
@T
@BEG_Attrib
3 @RT(0) @RT(16)cycle time in ms @RT(0)
@END_Attrib
1 0 @F @F @F @F

@Var @RT(9)bInitDone @RT(0) @T @F @DT @RT(4)BOOL @RT(0) @T @T @BASIC 0 @F
@F @F
@T
@BEG_Attrib
3 @RT(0) @RT(0) @RT(0)
@END_Attrib
1 0 @F @F @F @F

@Var @RT(14)rTaskCycleTime @RT(0) @T @F @DT @RT(4)REAL @RT(0) @T @T @BASIC 0 @F
@F @F
@T
@BEG_Attrib
3 @RT(0) @RT(0) @RT(0)
@END_Attrib
1 0 @F @F @F @F

@END_Dcl

@END_Export

@BEG_Body
@TL(32)
(**************************************** WARNING ********************************************
 *** The KEBA Kemro K2 System including software is not intended for safety control tasks! ***
 ***                       For further information see Comment tab!                        ***
 *********************************************************************************************)

IF NOT bInitDone THEN
   dTaskCycleTime := GET_TASK_INTERVAL();
   rTaskCycleTime := LINT_TO_REAL(TIME_TO_LINT(dTaskCycleTime)) / 1000000.0;   //task cycle time in sec
   bInitDone := TRUE;
END_IF;

rStepWidth := 2.0 * cApplPlasticsPI * rFrequency * rTaskCycleTime;

rOut := rAmplitude * SIN(rX);
rX := rX + rStepWidth;
IF rX > (2.0 * cApplPlasticsPI) THEN
    rX := rX - (2.0 * cApplPlasticsPI);
END_IF;

@END_Body

@END_Contents

(* ---- FBStandStill.pu ---- *)
(*
/*-------------------------------------------------------------------------
 *                   (c) 2002 by KEBA Ges.m.b.H & Co
 *                            Linz/AUSTRIA
 *                         All rights reserved
 *--------------------------------------------------------------------------
 *    Projekt   : moldmachine - demoapplication
 *    Erstautor : fal
 *    Datum     : 27.03.2003
 *    $Author: Fal $
 *    $Revision: 1 $
 *    $Modtime: 28.11.06 17:13 $
 *    $Archive: /ApplicationFrames/KePlast/APPL/ApplMoldMachineIECBase/FBStandStill.pu $
 *--------------------------------------------------------------------------*/
*)

IMPORT_OVER_LISTFILE
 TON

END_IMPORT

FUNCTION_BLOCK FBStandStill #DUMMY_EDIT_BLOCK

VAR_INPUT
 rActVoltage : REAL;
END_VAR

VAR_OUTPUT
 bStandStill : BOOL;
END_VAR

VAR_INPUT
 bDoCalib : BOOL;
 dCalibTime : TIME;
 rMaxVoltageDiff : REAL;
 dDelayTime : TIME;
END_VAR

VAR
 rVoltageTemp : REAL;
 rVoltageDifference : REAL;
 fbTON_Calib : TON;
 fbTON_Delay : TON;
END_VAR

(* IecGraph-Code *)

(* init step *)
INITIAL_STEP S_Init:
AInit (P);
END_STEP

ACTION AInit: #BEGIN_EDIT_BLOCK
fbTON_Calib(IN := FALSE, PT := dCalibTime);
fbTON_Delay(IN := FALSE, PT := dDelayTime);
bStandStill := FALSE;

;#END_EDIT_BLOCK END_ACTION (*AInit*)

(* steps *)
STEP S_Wait_PumpDelay:
ATimerDelay (N);
END_STEP

ACTION ATimerDelay: #BEGIN_EDIT_BLOCK
fbTON_Delay(IN := TRUE, PT := dDelayTime);

;#END_EDIT_BLOCK END_ACTION (*ATimerDelay*)
STEP S_SaveVoltage:
ATimer (N);
ASaveVoltage (P);
END_STEP

ACTION ATimer: #BEGIN_EDIT_BLOCK
fbTON_Calib(IN := TRUE, PT := dCalibTime);

;#END_EDIT_BLOCK END_ACTION (*ATimer*)
ACTION ASaveVoltage: #BEGIN_EDIT_BLOCK
rVoltageTemp := rActVoltage;

;#END_EDIT_BLOCK END_ACTION (*ASaveVoltage*)
STEP S_CalcDiff:
ACalcDiff (P);
END_STEP

ACTION ACalcDiff: #BEGIN_EDIT_BLOCK
rVoltageDifference := (ABS(rVoltageTemp - rActVoltage));
fbTON_Calib(IN := FALSE, PT := dCalibTime);

;#END_EDIT_BLOCK END_ACTION (*ACalcDiff*)
STEP S_StandStill:
AStandStill (P);
END_STEP

ACTION AStandStill: #BEGIN_EDIT_BLOCK
bStandStill := TRUE;

;#END_EDIT_BLOCK END_ACTION (*AStandStill*)

(* transitions *)
TRANSITION TStartCalib (* TStartCalib *) FROM S_Init TO S_Wait_PumpDelay :=  #BEGIN_EDIT_BLOCK
bDoCalib
;#END_EDIT_BLOCK
END_TRANSITION

TRANSITION Trans11 (* Trans11 *) FROM S_Wait_PumpDelay TO S_SaveVoltage :=  #BEGIN_EDIT_BLOCK
fbTON_Delay.Q
;#END_EDIT_BLOCK
END_TRANSITION

TRANSITION TCalcDifference (* TCalcDifference *) FROM S_SaveVoltage TO S_CalcDiff :=  #BEGIN_EDIT_BLOCK
fbTON_Calib.Q
;#END_EDIT_BLOCK
END_TRANSITION

TRANSITION TContinue (* TContinue *) FROM S_CalcDiff TO S_SaveVoltage :=  #BEGIN_EDIT_BLOCK
rVoltageDifference > rMaxVoltageDiff
;#END_EDIT_BLOCK
END_TRANSITION

TRANSITION TStandStillDetected (* TStandStillDetected *) FROM S_CalcDiff TO S_StandStill :=  #BEGIN_EDIT_BLOCK
rVoltageDifference <= rMaxVoltageDiff
;#END_EDIT_BLOCK
END_TRANSITION

TRANSITION TTrue (* TTrue *) FROM S_StandStill TO S_Init :=  #BEGIN_EDIT_BLOCK
TRUE
;#END_EDIT_BLOCK
END_TRANSITION

(* end IecGraph-Code *)
(* sfc-code *)

(* exits *)

EXIT_TRANSITION S_Stop := #BEGIN_EDIT_BLOCK
NOT bDoCalib
;#END_EDIT_BLOCK
PRIORITY 1 WITH  INITIAL_STEP S_Init: END_STEP
END_TRANSITION
(* end sfc-code *)

END_FUNCTION_BLOCK

#END_OF_IEC_PART

@Puma @IecEditor 6 113 @Pou 25
@@@BEG_Comment@@@
/*-------------------------------------------------------------------------
 *                   (c) 2002 by KEBA Ges.m.b.H & Co
 *                            Linz/AUSTRIA
 *                         All rights reserved
 *--------------------------------------------------------------------------
 *    Projekt   : moldmachine - demoapplication
 *    Erstautor : fal
 *    Datum     : 27.03.2003
 *    $Author: Fal $
 *    $Revision: 1 $
 *    $Modtime: 28.11.06 17:13 $
 *    $Archive: /ApplicationFrames/KePlast/APPL/ApplMoldMachineIECBase/FBStandStill.pu $
 *--------------------------------------------------------------------------*/
@@@END_Comment@@@

@BEG_Contents

@BEG_Func
@RT(17)FuncTreeContainer
0
@END_Func

@BEG_Const
@RT(18)ConstTreeContainer
0
@END_Const

@BEG_Export

@BEG_Kind
@FUNCTION_BLOCK @RT(12)FBStandStill @SEQUENTIAL_FLOW_CHART
@RT(0) @RT(0) @RT(0)
@END_Kind

@BEG_Dcl
@RT(16)DclTreeContainer
10
@Var @RT(11)rActVoltage @RT(0) @T @F @DT @RT(4)REAL @RT(0) @T @T @BASIC 0 @F
@F @F
@T
@BEG_Attrib
3 @RT(0) @RT(0) @RT(0)
@END_Attrib
1 1 @F @F @F @F

@Var @RT(11)bStandStill @RT(0) @T @F @DT @RT(4)BOOL @RT(0) @T @T @BASIC 0 @F
@F @F
@T
@BEG_Attrib
3 @RT(0) @RT(0) @RT(0)
@END_Attrib
1 3 @F @F @F @F

@Var @RT(8)bDoCalib @RT(0) @T @F @DT @RT(4)BOOL @RT(0) @T @T @BASIC 0 @F
@F @F
@T
@BEG_Attrib
3 @RT(0) @RT(0) @RT(0)
@END_Attrib
1 1 @F @F @F @F

@Var @RT(10)dCalibTime @RT(0) @T @F @DT @RT(4)TIME @RT(0) @T @T @BASIC 0 @F
@F @F
@T
@BEG_Attrib
3 @RT(0) @RT(0) @RT(0)
@END_Attrib
1 1 @F @F @F @F

@Var @RT(15)rMaxVoltageDiff @RT(0) @T @F @DT @RT(4)REAL @RT(0) @T @T @BASIC 0 @F
@F @F
@T
@BEG_Attrib
3 @RT(0) @RT(0) @RT(0)
@END_Attrib
1 1 @F @F @F @F

@Var @RT(10)dDelayTime @RT(0) @T @F @DT @RT(4)TIME @RT(0) @T @T @BASIC 0 @F
@F @F
@T
@BEG_Attrib
3 @RT(0) @RT(0) @RT(0)
@END_Attrib
1 1 @F @F @F @F

@Var @RT(12)rVoltageTemp @RT(0) @T @F @DT @RT(4)REAL @RT(0) @T @T @BASIC 0 @F
@F @F
@T
@BEG_Attrib
3 @RT(0) @RT(0) @RT(0)
@END_Attrib
1 0 @F @F @F @F

@Var @RT(18)rVoltageDifference @RT(0) @T @F @DT @RT(4)REAL @RT(0) @T @T @BASIC 0 @F
@F @F
@T
@BEG_Attrib
3 @RT(0) @RT(0) @RT(0)
@END_Attrib
1 0 @F @F @F @F

@Var @RT(11)fbTON_Calib @RT(0) @T @T @DERIVED 0 @T @T @DT @RT(3)TON @RT(0) @T @T @UNKNOWN 0 @F
@F @F
@T
@BEG_Attrib
3 @RT(0) @RT(0) @RT(0)
@END_Attrib
1 0 @F @F @F @F

@Var @RT(11)fbTON_Delay @RT(0) @T @T @DERIVED 0 @T @T @DT @RT(3)TON @RT(0) @T @T @UNKNOWN 0 @F
@F @F
@T
@BEG_Attrib
3 @RT(0) @RT(0) @RT(0)
@END_Attrib
1 0 @F @F @F @F

@END_Dcl

@END_Export

@BEG_SfcBody
7 7 7

@BEG_SfcData 2
@StepSeq @RT(4)sseq @F 9
@Step @RT(6)S_Init @F @T @T @F @RT(0) @F
@AcbCont @RT(7)unnamed @F 1
@Acb @RT(5)AInit @F @T @RT(1)P @RT(0) @F @F @T @TL(4)
fbTON_Calib(IN := FALSE, PT := dCalibTime);
fbTON_Delay(IN := FALSE, PT := dDelayTime);
bStandStill := FALSE;

@F

@Trans @RT(11)TStartCalib @F @T @F @F @T @T @TL(2)
bDoCalib

@RT(11)TStartCalib @F
@Step @RT(16)S_Wait_PumpDelay @F @F @F @F @RT(0) @F
@AcbCont @RT(7)unnamed @F 1
@Acb @RT(11)ATimerDelay @F @T @RT(1)N @RT(0) @F @F @T @TL(2)
fbTON_Delay(IN := TRUE, PT := dDelayTime);

@F

@Trans @RT(7)Trans11 @F @T @F @F @T @T @TL(2)
fbTON_Delay.Q

@RT(7)Trans11 @F
@Loop @RT(4)loop @F 2
@StepSeq @RT(4)sseq @F 3
@Step @RT(13)S_SaveVoltage @F @F @F @F @RT(0) @F
@AcbCont @RT(7)unnamed @F 2
@Acb @RT(6)ATimer @F @T @RT(1)N @RT(0) @F @F @T @TL(2)
fbTON_Calib(IN := TRUE, PT := dCalibTime);

@F
@Acb @RT(12)ASaveVoltage @F @T @RT(1)P @RT(0) @F @F @T @TL(2)
rVoltageTemp := rActVoltage;

@F

@Trans @RT(15)TCalcDifference @F @T @F @F @T @T @TL(2)
fbTON_Calib.Q

@RT(15)TCalcDifference @F
@Step @RT(10)S_CalcDiff @F @F @F @F @RT(0) @F
@AcbCont @RT(7)unnamed @F 1
@Acb @RT(9)ACalcDiff @F @T @RT(1)P @RT(0) @F @F @T @TL(3)
rVoltageDifference := (ABS(rVoltageTemp - rActVoltage));
fbTON_Calib(IN := FALSE, PT := dCalibTime);

@F

@Trans @RT(9)TContinue @F @T @F @T @T @T @TL(2)
rVoltageDifference > rMaxVoltageDiff

@RT(9)TContinue @F

@Trans @RT(19)TStandStillDetected @F @T @F @F @T @T @TL(2)
rVoltageDifference <= rMaxVoltageDiff

@RT(19)TStandStillDetected @F
@Step @RT(12)S_StandStill @F @F @F @F @RT(0) @F
@AcbCont @RT(7)unnamed @F 1
@Acb @RT(11)AStandStill @F @T @RT(1)P @RT(0) @F @F @T @TL(2)
bStandStill := TRUE;

@F

@Trans @RT(5)TTrue @F @T @F @F @T @T @TL(2)
TRUE

@RT(5)TTrue @F
@Goto @RT(6)S_Init @F @F
@END_SfcData
@SaActions 0
@SaTrans 0
@SaExits 1
@SaExit @SaText @RT(6)S_Stop 1 @TL(2)
NOT bDoCalib

@RT(6)S_Init @RT(1)1 @F @F @SaSfc @RT(6)S_Stop 5 @RT(5)DUMMY
@BEG_SfcData 2
@ExitSeq @RT(4)sseq @F 3
@Step @RT(8)unnamed1 @F @T @F @F @RT(0) @F
@AcbCont @RT(7)unnamed @F 0

@Trans @RT(8)unnamed3 @F @T @F @F @T @T @TL(2)

@RT(8)unnamed3 @F
@Goto @RT(9)unlabeled @F @F
@END_SfcData

@END_SfcBody

@END_Contents
